# B&R Automation Studio project RobotComau
Automation Studio 4.11.2.75; technology packages: mapp 5.18.0, mappMotion 5.18.1, mappView 5.18.1, mappVision 5.18.0

## Configuration Config1

CPU 5APC3100.KBU1-000, AutomationRuntime B4.92, Build 4.1.2, Safety 0.0, Vc V4.72.5

### Task classes (Cpu.sw)
```
Cyclic#1 (cycle 2000 us, tolerance 0 us):
  Comau <- Comau.prg [disabled]
  OpcCtrl <- Sources.OpcCtrl.prg
  ComauManua <- PackML.PackML_Manual.prg
  PackML_Aut <- PackML.PackML_Auto.prg
  PackML_Log <- PackML.PackML_Logic.prg
  PackML_Sem <- PackML.PackML_SemiAuto.prg
  RobotMove <- (binary)
Cyclic#4:
  Alarms <- Alarms.prg
  Elements_d <- Elements_detection.prg
DataObjects: McAcpSys
NcDataObjects: McDriveLog
Binaries: McAcpDrv, udbdef, McAcpSim, mvLoader, arflatprv, McPathXT, TCData, visionUnit, mCoWebSc, McMechSys, FWRules, arcoal, arsvcreg, Settings, iomap, Config_3, Settings_1, viComp, Config_4, Role, ashwac, Hierarchy, asfw, Config_5, sysconf, Config_2, arconfig, Config_1, ashwd, User, Config_6, Config, Config_7, Config_9, PixelCount, Config_8, viApp, Matching15
Libraries: McBase, ViBase, AsZip, FileIO, AsARCfg, powerlnk, AsEPL, AsIO, sys_lib, astime, runtime, MpRobotics, McAxGroup, MpBase, McPathGen, McAxis, McProgInt, McAcpAx, CoTrace, standard, MpPackML, MpAlarmX, MpServer, MpUserX, asarprof, asieccon, asarlog, asmem, brsystem, dataobj, arssl, asopcuac, aseth, ashw, arcert, aruser
```

### Hardware
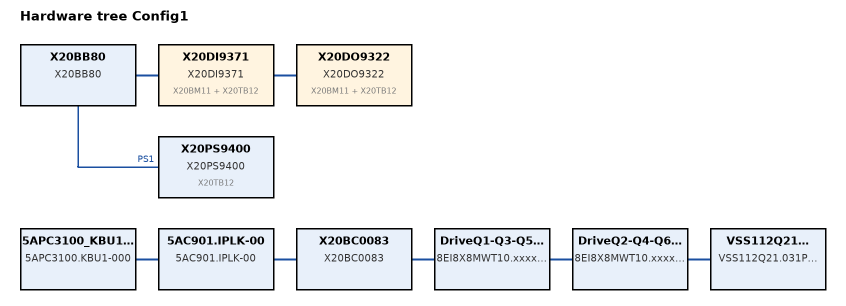
```
5AC901.IPLK-00 : 5AC901.IPLK-00 v1.8.0.1  [SL -> 5APC3100_KBU1_000.SL2]
  Connector IF1:
    MtuSize = 1500
    CycleTime = 400
    Channel1
    ChannelID1 = McAcpBroadcast
    ChannelType1 = OCTET[200]
    InternetAddress = 192.168.200.240
    SubnetMask = 255.255.255.0
5APC3100_KBU1_000 : 5APC3100.KBU1-000 v2.2.1.0
  Connector IF3:
    AssignedOperatingSystem = ARemb
    ActivateDevice = 1
    Mode = Manual
    InternetAddress = 192.168.0.10
    SubnetMask = 255.255.255.0
    ActivateSnmp = 2
  Connector IF4:
    AssignedOperatingSystem = ARemb
    ActivateDevice = 1
  Connector IF5:
    AssignedOperatingSystem = ARemb
  Connector IF6:
    AssignedOperatingSystem = ARemb
  Connector IF7:
    AssignedOperatingSystem = ARemb
  Connector IF8:
    AssignedOperatingSystem = ARemb
  ConfigurationID = RobotComau_Config1
  Simulation = 1
  RemMemDevice = PCI.2.IPLK.SRAM
  RemMemSize = 1024
  PermanentPvSize = 512
  RemanentGlobalPvSize = 512
  TimerDeviceType = EPLX2X
  TimerDevice = 5AC901.IPLK-00.IF1
  TaskClassIdleTime = 2000
  Cyclic1Duration = 2000
  Cyclic1Tolerance = 0
  FileDevice1
  FileDeviceName1 = CNC_PrgDir
  FileDevicePath1 = F:\RobotProgram
  FileDevice2
  FileDeviceName2 = F
  FileDevicePath2 = F:\
  FtpUser1
  FtpUsername1 = admin
  FtpUserPassword1 = QCzPEyxrRcQJkbJUmFYJydudCaTwVAMxyUFRcNQN44M=
  FtpUserSalt1 = 07CFXo9y
  FTPAccessRight1 = 0
  ActivateOpcUa = 1
  OpcUaInformationModels_PV_Version = 1
DriveQ1-Q3-Q5_Racer3_1 : 8EI8X8MWT10.xxxx-1 v2.3.1.1  [PLK1 -> X20BC0083.PLK2 (NodeNumber=4) [Cable Type=PowerlinkCable, Length=10, Version=1.0.0.3]; PLK2 -> DriveQ2-Q4-Q6_Racer3_1.PLK1 (NodeNumber=4) [Cable Type=PowerlinkCable, Length=10, Version=1.0.0.3]]
  DriveConfiguration/Module:
    McAcoposTypeID = AcoposP3TConfig
    ActivateACOPOSSimulationOnPLC = 0
  DriveConfiguration/Encoder/EncoderX41:
    InterfaceType = EnDat
  DriveConfiguration/Encoder/EncoderX42:
    InterfaceType = EnDat
  DriveConfiguration/Encoder/EncoderX43:
    InterfaceType = EnDat
  DriveConfiguration/Channel[1]/RealAxis:
    AxisReference = gAxisQ1_Racer3_1
    MechanicalElementsIsInvisible = 0
  DriveConfiguration/Channel[1]/RealAxis/MechanicalElements/Gearbox:
    InputIsReadOnly = 1
    Input = 81818
    OutputIsReadOnly = 1
    Output = 1000
  DriveConfiguration/Channel[1]/RealAxis/MechanicalElements/RotaryToLinearTransformation:
    ReferenceDistanceIsReadOnly = 1
    ReferenceDistance = 360
  DriveConfiguration/Channel[1]/RealAxis/Controller:
    ModeIsReadOnly = 1
    Mode = PositionControllerWithTorqueFeedForward
  DriveConfiguration/Channel[1]/RealAxis/Controller/Mode/Position:
    ProportionalGainIsReadOnly = 1
    ProportionalGain = 75.0
    IntegrationTimeIsReadOnly = 1
    IntegrationTime = 0.0
    TotalDelayTime = 0.0004
  DriveConfiguration/Channel[1]/RealAxis/Controller/Mode/Speed:
    ProportionalGainIsReadOnly = 1
    ProportionalGain = 2.0
    IntegrationTimeIsReadOnly = 1
    IntegrationTime = 0.0
    FilterTimeIsReadOnly = 1
    FilterTime = 0.0008
  DriveConfiguration/Channel[1]/RealAxis/Controller/Mode:
    FeedForwardIsReadOnly = 1
    FeedForward = CyclicValueFromAxesGroup
  DriveConfiguration/Channel[1]/RealAxis/Controller/Mode/LoopFilters:
    LoopFilterXIsReadOnly = 0
    LoopFilter1 = NotUsed
    LoopFilter2 = NotUsed
    LoopFilter3 = NotUsed
  DriveConfiguration/Channel[1]/RealAxis/Homing:
    ModeIsReadOnly = 0
    Mode = RestorePosition
    RestorePositionVariable = ::RestorePos[0]
  DriveConfiguration/Channel[1]/RealAxis/StopReaction:
    QuickstopIsReadOnly = 0
    Quickstop = DecelerationLimit
    DriveErrorIsReadOnly = 0
    DriveError = DecelerationLimit
  DriveConfiguration/Channel[1]/RealAxis/MovementErrorLimits:
    PositionError = 1.0
    VelocityErrorMonitoring = Automatic1
  DriveConfiguration/Channel[1]/RealAxis:
    JerkFilterIsReadOnly = 0
    JerkFilter = Used
  DriveConfiguration/Channel[1]/RealAxis/JerkFilter:
    JerkTimeMin = 0
    JerkTime = 0.01
  DriveConfiguration/Channel[1]/RealAxis/DigitalInputs/HomingSwitch:
    SourceIsReadOnly = 0
    Source = NotUsed
    Level = High
  DriveConfiguration/Channel[1]/RealAxis/DigitalInputs/PositiveLimitSwitch:
    SourceIsReadOnly = 0
    Source = NotUsed
    Level = High
  DriveConfiguration/Channel[1]/RealAxis/DigitalInputs/NegativeLimitSwitch:
    SourceIsReadOnly = 0
    Source = NotUsed
    Level = High
  DriveConfiguration/Channel[1]/RealAxis/DigitalInputs/Trigger1:
    Source = X8Trigger1
    Level = High
  DriveConfiguration/Channel[1]/RealAxis/DigitalInputs/Trigger2:
    Source = X8Trigger2
    Level = High
  DriveConfiguration/Channel[1]/RealAxis/DigitalInputs/Quickstop:
    Input = Trigger2
  DriveConfiguration/Channel[1]/RealAxis/Simulation:
    SimulationModeOnPLC = SetValueGeneration
    SimulationModeOnACOPOS = NotUsed
  DriveConfiguration/Channel[1]/RealAxis/AxisFeatures:
    FeatureRef[1] = Feature_Brake_Racer3_1
  DriveConfiguration/Channel[1]:
    ExternalEncoderAxis = NotUsed
  DriveConfiguration/Channel[2]/RealAxis:
    AxisReference = gAxisQ3_Racer3_1
    MechanicalElementsIsInvisible = 0
  DriveConfiguration/Channel[2]/RealAxis/MechanicalElements/Gearbox:
    InputIsReadOnly = 1
    Input = 72
    OutputIsReadOnly = 1
    Output = 1
  DriveConfiguration/Channel[2]/RealAxis/MechanicalElements/RotaryToLinearTransformation:
    ReferenceDistanceIsReadOnly = 1
    ReferenceDistance = 360
  DriveConfiguration/Channel[2]/RealAxis/Controller:
    ModeIsReadOnly = 1
    Mode = PositionControllerWithTorqueFeedForward
  DriveConfiguration/Channel[2]/RealAxis/Controller/Mode/Position:
    ProportionalGainIsReadOnly = 1
    ProportionalGain = 50.0
    IntegrationTimeIsReadOnly = 1
    IntegrationTime = 0.0
    TotalDelayTime = 0.0004
  DriveConfiguration/Channel[2]/RealAxis/Controller/Mode/Speed:
    ProportionalGainIsReadOnly = 1
    ProportionalGain = 1.5
    IntegrationTimeIsReadOnly = 1
    IntegrationTime = 0.0
    FilterTimeIsReadOnly = 1
    FilterTime = 0.0008
  DriveConfiguration/Channel[2]/RealAxis/Controller/Mode:
    FeedForwardIsReadOnly = 1
    FeedForward = CyclicValueFromAxesGroup
  DriveConfiguration/Channel[2]/RealAxis/Controller/Mode/LoopFilters:
    LoopFilterXIsReadOnly = 0
    LoopFilter1 = NotUsed
    LoopFilter2 = NotUsed
    LoopFilter3 = NotUsed
  DriveConfiguration/Channel[2]/RealAxis/Homing:
    ModeIsReadOnly = 0
    Mode = RestorePosition
    RestorePositionVariable = ::RestorePos[2]
  DriveConfiguration/Channel[2]/RealAxis/StopReaction:
    QuickstopIsReadOnly = 0
    Quickstop = DecelerationLimit
    DriveErrorIsReadOnly = 0
    DriveError = DecelerationLimit
  DriveConfiguration/Channel[2]/RealAxis/MovementErrorLimits:
    PositionError = 1.0
    VelocityErrorMonitoring = Automatic1
  DriveConfiguration/Channel[2]/RealAxis:
    JerkFilterIsReadOnly = 0
    JerkFilter = Used
  DriveConfiguration/Channel[2]/RealAxis/JerkFilter:
    JerkTimeMin = 0
    JerkTime = 0.01
  DriveConfiguration/Channel[2]/RealAxis/DigitalInputs/HomingSwitch:
    SourceIsReadOnly = 0
    Source = NotUsed
    Level = High
  DriveConfiguration/Channel[2]/RealAxis/DigitalInputs/PositiveLimitSwitch:
    SourceIsReadOnly = 0
    Source = NotUsed
    Level = High
  DriveConfiguration/Channel[2]/RealAxis/DigitalInputs/NegativeLimitSwitch:
    SourceIsReadOnly = 0
    Source = NotUsed
    Level = High
  DriveConfiguration/Channel[2]/RealAxis/DigitalInputs/Trigger1:
    Source = X8Trigger1
    Level = High
  DriveConfiguration/Channel[2]/RealAxis/DigitalInputs/Trigger2:
    Source = X8Trigger2
    Level = High
  DriveConfiguration/Channel[2]/RealAxis/DigitalInputs/Quickstop:
    Input = Trigger2
  DriveConfiguration/Channel[2]/RealAxis/Simulation:
    SimulationModeOnPLC = SetValueGeneration
    SimulationModeOnACOPOS = NotUsed
  DriveConfiguration/Channel[2]/RealAxis/AxisFeatures:
    FeatureRef[1] = Feature_Brake_Racer3_1
  DriveConfiguration/Channel[2]:
    ExternalEncoderAxis = NotUsed
  DriveConfiguration/Channel[3]/RealAxis:
    AxisReference = gAxisQ5_Racer3_1
    MechanicalElementsIsInvisible = 0
  DriveConfiguration/Channel[3]/RealAxis/MechanicalElements/Gearbox:
    InputIsReadOnly = 1
    Input = 612
    OutputIsReadOnly = 1
    Output = 10
  DriveConfiguration/Channel[3]/RealAxis/MechanicalElements/RotaryToLinearTransformation:
    ReferenceDistanceIsReadOnly = 1
    ReferenceDistance = 360
  DriveConfiguration/Channel[3]/RealAxis/Controller:
    ModeIsReadOnly = 1
    Mode = PositionControllerWithTorqueFeedForward
  DriveConfiguration/Channel[3]/RealAxis/Controller/Mode/Position:
    ProportionalGainIsReadOnly = 1
    ProportionalGain = 200.0
    IntegrationTimeIsReadOnly = 1
    IntegrationTime = 0.0
    TotalDelayTime = 0.0004
  DriveConfiguration/Channel[3]/RealAxis/Controller/Mode/Speed:
    ProportionalGainIsReadOnly = 1
    ProportionalGain = 1.5
    IntegrationTimeIsReadOnly = 1
    IntegrationTime = 0.0
    FilterTimeIsReadOnly = 1
    FilterTime = 0.0008
  DriveConfiguration/Channel[3]/RealAxis/Controller/Mode:
    FeedForwardIsReadOnly = 1
    FeedForward = CyclicValueFromAxesGroup
  DriveConfiguration/Channel[3]/RealAxis/Controller/Mode/LoopFilters:
    LoopFilterXIsReadOnly = 0
    LoopFilter1 = NotUsed
    LoopFilter2 = NotUsed
    LoopFilter3 = NotUsed
  DriveConfiguration/Channel[3]/RealAxis/Homing:
    ModeIsReadOnly = 0
    Mode = RestorePosition
    RestorePositionVariable = ::RestorePos[4]
  DriveConfiguration/Channel[3]/RealAxis/StopReaction:
    QuickstopIsReadOnly = 0
    Quickstop = DecelerationLimit
    DriveErrorIsReadOnly = 0
    DriveError = DecelerationLimit
  DriveConfiguration/Channel[3]/RealAxis/MovementErrorLimits:
    PositionError = 1.0
    VelocityErrorMonitoring = Automatic1
  DriveConfiguration/Channel[3]/RealAxis:
    JerkFilterIsReadOnly = 0
    JerkFilter = Used
  DriveConfiguration/Channel[3]/RealAxis/JerkFilter:
    JerkTimeMin = 0
    JerkTime = 0.01
  DriveConfiguration/Channel[3]/RealAxis/DigitalInputs/HomingSwitch:
    SourceIsReadOnly = 0
    Source = NotUsed
    Level = High
  DriveConfiguration/Channel[3]/RealAxis/DigitalInputs/PositiveLimitSwitch:
    SourceIsReadOnly = 0
    Source = NotUsed
    Level = High
  DriveConfiguration/Channel[3]/RealAxis/DigitalInputs/NegativeLimitSwitch:
    SourceIsReadOnly = 0
    Source = NotUsed
    Level = High
  DriveConfiguration/Channel[3]/RealAxis/DigitalInputs/Trigger1:
    Source = X8Trigger1
    Level = High
  DriveConfiguration/Channel[3]/RealAxis/DigitalInputs/Trigger2:
    Source = X8Trigger2
    Level = High
  DriveConfiguration/Channel[3]/RealAxis/DigitalInputs/Quickstop:
    Input = Trigger2
  DriveConfiguration/Channel[3]/RealAxis/Simulation:
    SimulationModeOnPLC = SetValueGeneration
    SimulationModeOnACOPOS = NotUsed
  DriveConfiguration/Channel[3]/RealAxis/AxisFeatures:
    FeatureRef[1] = Feature_Brake_Racer3_1
  DriveConfiguration/Channel[3]:
    ExternalEncoderAxis = NotUsed
DriveQ2-Q4-Q6_Racer3_1 : 8EI8X8MWT10.xxxx-1 v2.3.1.1  [PLK1 -> DriveQ1-Q3-Q5_Racer3_1.PLK2 (NodeNumber=5) [Cable Type=PowerlinkCable, Length=10, Version=1.0.0.3]; PLK2 -> VSS112Q21.031P-000.PLK2 (NodeNumber=5) [Cable Type=PowerlinkCable, Length=10, Version=1.0.0.3]]
  DriveConfiguration/Module:
    McAcoposTypeID = AcoposP3TConfig
    ActivateACOPOSSimulationOnPLC = 0
  DriveConfiguration/Encoder/EncoderX41:
    InterfaceType = EnDat
  DriveConfiguration/Encoder/EncoderX42:
    InterfaceType = EnDat
  DriveConfiguration/Encoder/EncoderX43:
    InterfaceType = EnDat
  DriveConfiguration/Channel[1]/RealAxis:
    AxisReference = gAxisQ2_Racer3_1
    MechanicalElementsIsInvisible = 0
  DriveConfiguration/Channel[1]/RealAxis/MechanicalElements/Gearbox:
    InputIsReadOnly = 1
    Input = 80
    OutputIsReadOnly = 1
    Output = 1
  DriveConfiguration/Channel[1]/RealAxis/MechanicalElements/RotaryToLinearTransformation:
    ReferenceDistanceIsReadOnly = 1
    ReferenceDistance = 360
  DriveConfiguration/Channel[1]/RealAxis/Controller:
    ModeIsReadOnly = 1
    Mode = PositionControllerWithTorqueFeedForward
  DriveConfiguration/Channel[1]/RealAxis/Controller/Mode/Position:
    ProportionalGainIsReadOnly = 1
    ProportionalGain = 50.0
    IntegrationTimeIsReadOnly = 1
    IntegrationTime = 0.0
    TotalDelayTime = 0.0004
  DriveConfiguration/Channel[1]/RealAxis/Controller/Mode/Speed:
    ProportionalGainIsReadOnly = 1
    ProportionalGain = 2.0
    IntegrationTimeIsReadOnly = 1
    IntegrationTime = 0.0
    FilterTimeIsReadOnly = 1
    FilterTime = 0.0008
  DriveConfiguration/Channel[1]/RealAxis/Controller/Mode:
    FeedForwardIsReadOnly = 1
    FeedForward = CyclicValueFromAxesGroup
  DriveConfiguration/Channel[1]/RealAxis/Controller/Mode/LoopFilters:
    LoopFilterXIsReadOnly = 0
    LoopFilter1 = NotUsed
    LoopFilter2 = NotUsed
    LoopFilter3 = NotUsed
  DriveConfiguration/Channel[1]/RealAxis/Homing:
    ModeIsReadOnly = 0
    Mode = RestorePosition
    RestorePositionVariable = ::RestorePos[1]
  DriveConfiguration/Channel[1]/RealAxis/StopReaction:
    QuickstopIsReadOnly = 0
    Quickstop = DecelerationLimit
    DriveErrorIsReadOnly = 0
    DriveError = DecelerationLimit
  DriveConfiguration/Channel[1]/RealAxis/MovementErrorLimits:
    PositionError = 1.0
    VelocityErrorMonitoring = Automatic1
  DriveConfiguration/Channel[1]/RealAxis:
    JerkFilterIsReadOnly = 0
    JerkFilter = Used
  DriveConfiguration/Channel[1]/RealAxis/JerkFilter:
    JerkTimeMin = 0
    JerkTime = 0.01
  DriveConfiguration/Channel[1]/RealAxis/DigitalInputs/HomingSwitch:
    SourceIsReadOnly = 0
    Source = NotUsed
    Level = High
  DriveConfiguration/Channel[1]/RealAxis/DigitalInputs/PositiveLimitSwitch:
    SourceIsReadOnly = 0
    Source = NotUsed
    Level = High
  DriveConfiguration/Channel[1]/RealAxis/DigitalInputs/NegativeLimitSwitch:
    SourceIsReadOnly = 0
    Source = NotUsed
    Level = High
  DriveConfiguration/Channel[1]/RealAxis/DigitalInputs/Trigger1:
    Source = X8Trigger1
    Level = High
  DriveConfiguration/Channel[1]/RealAxis/DigitalInputs/Trigger2:
    Source = X8Trigger2
    Level = High
  DriveConfiguration/Channel[1]/RealAxis/DigitalInputs/Quickstop:
    Input = Trigger2
  DriveConfiguration/Channel[1]/RealAxis/Simulation:
    SimulationModeOnPLC = SetValueGeneration
    SimulationModeOnACOPOS = NotUsed
  DriveConfiguration/Channel[1]/RealAxis/AxisFeatures:
    FeatureRef[1] = Feature_Brake_Racer3_1
  DriveConfiguration/Channel[1]:
    ExternalEncoderAxis = NotUsed
  DriveConfiguration/Channel[2]/RealAxis:
    AxisReference = gAxisQ4_Racer3_1
    MechanicalElementsIsInvisible = 0
  DriveConfiguration/Channel[2]/RealAxis/MechanicalElements/Gearbox:
    InputIsReadOnly = 1
    Input = 612
    OutputIsReadOnly = 1
    Output = 10
  DriveConfiguration/Channel[2]/RealAxis/MechanicalElements/RotaryToLinearTransformation:
    ReferenceDistanceIsReadOnly = 1
    ReferenceDistance = 360
  DriveConfiguration/Channel[2]/RealAxis/Controller:
    ModeIsReadOnly = 1
    Mode = PositionControllerWithTorqueFeedForward
  DriveConfiguration/Channel[2]/RealAxis/Controller/Mode/Position:
    ProportionalGainIsReadOnly = 1
    ProportionalGain = 100.0
    IntegrationTimeIsReadOnly = 1
    IntegrationTime = 0.0
    TotalDelayTime = 0.0004
  DriveConfiguration/Channel[2]/RealAxis/Controller/Mode/Speed:
    ProportionalGainIsReadOnly = 1
    ProportionalGain = 2.0
    IntegrationTimeIsReadOnly = 1
    IntegrationTime = 0.0
    FilterTimeIsReadOnly = 1
    FilterTime = 0.0008
  DriveConfiguration/Channel[2]/RealAxis/Controller/Mode:
    FeedForwardIsReadOnly = 1
    FeedForward = CyclicValueFromAxesGroup
  DriveConfiguration/Channel[2]/RealAxis/Controller/Mode/LoopFilters:
    LoopFilterXIsReadOnly = 0
    LoopFilter1 = NotUsed
    LoopFilter2 = NotUsed
    LoopFilter3 = NotUsed
  DriveConfiguration/Channel[2]/RealAxis/Homing:
    ModeIsReadOnly = 0
    Mode = RestorePosition
    RestorePositionVariable = ::RestorePos[3]
  DriveConfiguration/Channel[2]/RealAxis/StopReaction:
    QuickstopIsReadOnly = 0
    Quickstop = DecelerationLimit
    DriveErrorIsReadOnly = 0
    DriveError = DecelerationLimit
  DriveConfiguration/Channel[2]/RealAxis/MovementErrorLimits:
    PositionError = 1.0
    VelocityErrorMonitoring = Automatic1
  DriveConfiguration/Channel[2]/RealAxis:
    JerkFilterIsReadOnly = 0
    JerkFilter = Used
  DriveConfiguration/Channel[2]/RealAxis/JerkFilter:
    JerkTimeMin = 0
    JerkTime = 0.01
  DriveConfiguration/Channel[2]/RealAxis/DigitalInputs/HomingSwitch:
    SourceIsReadOnly = 0
    Source = NotUsed
    Level = High
  DriveConfiguration/Channel[2]/RealAxis/DigitalInputs/PositiveLimitSwitch:
    SourceIsReadOnly = 0
    Source = NotUsed
    Level = High
  DriveConfiguration/Channel[2]/RealAxis/DigitalInputs/NegativeLimitSwitch:
    SourceIsReadOnly = 0
    Source = NotUsed
    Level = High
  DriveConfiguration/Channel[2]/RealAxis/DigitalInputs/Trigger1:
    Source = X8Trigger1
    Level = High
  DriveConfiguration/Channel[2]/RealAxis/DigitalInputs/Trigger2:
    Source = X8Trigger2
    Level = High
  DriveConfiguration/Channel[2]/RealAxis/DigitalInputs/Quickstop:
    Input = Trigger2
  DriveConfiguration/Channel[2]/RealAxis/Simulation:
    SimulationModeOnPLC = SetValueGeneration
    SimulationModeOnACOPOS = NotUsed
  DriveConfiguration/Channel[2]/RealAxis/AxisFeatures:
    FeatureRef[1] = Feature_Brake_Racer3_1
  DriveConfiguration/Channel[2]:
    ExternalEncoderAxis = NotUsed
  DriveConfiguration/Channel[3]/RealAxis:
    AxisReference = gAxisQ6_Racer3_1
    MechanicalElementsIsInvisible = 0
  DriveConfiguration/Channel[3]/RealAxis/MechanicalElements/Gearbox:
    InputIsReadOnly = 1
    Input = 40
    OutputIsReadOnly = 1
    Output = 1
  DriveConfiguration/Channel[3]/RealAxis/MechanicalElements/RotaryToLinearTransformation:
    ReferenceDistanceIsReadOnly = 1
    ReferenceDistance = 360
  DriveConfiguration/Channel[3]/RealAxis/Controller:
    ModeIsReadOnly = 1
    Mode = PositionControllerWithTorqueFeedForward
  DriveConfiguration/Channel[3]/RealAxis/Controller/Mode/Position:
    ProportionalGainIsReadOnly = 1
    ProportionalGain = 200.0
    IntegrationTimeIsReadOnly = 1
    IntegrationTime = 0.0
    TotalDelayTime = 0.0004
  DriveConfiguration/Channel[3]/RealAxis/Controller/Mode/Speed:
    ProportionalGainIsReadOnly = 1
    ProportionalGain = 1.5
    IntegrationTimeIsReadOnly = 1
    IntegrationTime = 0.0
    FilterTimeIsReadOnly = 1
    FilterTime = 0.0008
  DriveConfiguration/Channel[3]/RealAxis/Controller/Mode:
    FeedForwardIsReadOnly = 1
    FeedForward = CyclicValueFromAxesGroup
  DriveConfiguration/Channel[3]/RealAxis/Controller/Mode/LoopFilters:
    LoopFilterXIsReadOnly = 0
    LoopFilter1 = NotUsed
    LoopFilter2 = NotUsed
    LoopFilter3 = NotUsed
  DriveConfiguration/Channel[3]/RealAxis/Homing:
    ModeIsReadOnly = 0
    Mode = RestorePosition
    RestorePositionVariable = ::RestorePos[5]
  DriveConfiguration/Channel[3]/RealAxis/StopReaction:
    QuickstopIsReadOnly = 0
    Quickstop = DecelerationLimit
    DriveErrorIsReadOnly = 0
    DriveError = DecelerationLimit
  DriveConfiguration/Channel[3]/RealAxis/MovementErrorLimits:
    PositionError = 1.0
    VelocityErrorMonitoring = Automatic1
  DriveConfiguration/Channel[3]/RealAxis:
    JerkFilterIsReadOnly = 0
    JerkFilter = Used
  DriveConfiguration/Channel[3]/RealAxis/JerkFilter:
    JerkTimeMin = 0
    JerkTime = 0.01
  DriveConfiguration/Channel[3]/RealAxis/DigitalInputs/HomingSwitch:
    SourceIsReadOnly = 0
    Source = NotUsed
    Level = High
  DriveConfiguration/Channel[3]/RealAxis/DigitalInputs/PositiveLimitSwitch:
    SourceIsReadOnly = 0
    Source = NotUsed
    Level = High
  DriveConfiguration/Channel[3]/RealAxis/DigitalInputs/NegativeLimitSwitch:
    SourceIsReadOnly = 0
    Source = NotUsed
    Level = High
  DriveConfiguration/Channel[3]/RealAxis/DigitalInputs/Trigger1:
    Source = X8Trigger1
    Level = High
  DriveConfiguration/Channel[3]/RealAxis/DigitalInputs/Trigger2:
    Source = X8Trigger2
    Level = High
  DriveConfiguration/Channel[3]/RealAxis/DigitalInputs/Quickstop:
    Input = Trigger2
  DriveConfiguration/Channel[3]/RealAxis/Simulation:
    SimulationModeOnPLC = SetValueGeneration
    SimulationModeOnACOPOS = NotUsed
  DriveConfiguration/Channel[3]/RealAxis/AxisFeatures:
    FeatureRef[1] = Feature_Brake_Racer3_1
  DriveConfiguration/Channel[3]:
    ExternalEncoderAxis = NotUsed
VSS112Q21.031P-000 : VSS112Q21.031P-000 v1.6.0.543  [PLK2 -> DriveQ2-Q4-Q6_Racer3_1.PLK2 (NodeNumber=6) [Cable Type=PowerlinkCable, Length=10, Version=1.0.0.3]]
  VisionConfig = gCamera
X20BB80 : X20BB80 v1.1.0.0
X20BC0083 : X20BC0083 v2.12.0.0  [PLK1 -> 5AC901.IPLK-00.IF1 (NodeNumber=3) [Cable Type=PowerlinkCable, Length=10, Version=1.0.0.3]; PLK2 -> DriveQ1-Q3-Q5_Racer3_1.PLK1 (NodeNumber=3) [Cable Type=PowerlinkCable, Length=10, Version=1.0.0.3]; SL -> X20BB80.SL1]
X20BM11 : X20BM11 v1.1.0.0  [X2X1 -> X20BB80.IF1]
X20BM11a : X20BM11 v1.1.0.0  [X2X1 -> X20BM11.X2X2]
X20DI9371 : X20DI9371 v1.3.0.0  [SS1 -> X20TB12a.SS; SL -> X20BM11.SL1]
X20DO9322 : X20DO9322 v1.4.0.0  [SS1 -> X20TB12b.SS; SL -> X20BM11a.SL1]
X20PS9400 : X20PS9400 v1.7.0.0  [SS1 -> X20TB12.SS; PS -> X20BB80.PS1]
X20TB12 : X20TB12 v1.0.0.0
X20TB12a : X20TB12 v1.0.0.0
X20TB12b : X20TB12 v1.0.0.0
```

### IoMap.iom - 5APC3100_KBU1_000/IoMap.iom
```iecst
VAR_CONFIG
	::Elements_d:Camera_0.ImageAcq AT %QX."VSS112Q21.031P-000".ImageAcquisition;
	::Elements_d:Camera_0.PixelCntSquareArray[0] AT %ID."VSS112Q21.031P-000".FoundedPixelsNum01;
	::Elements_d:Camera_0.PixelCntSquareArray[1] AT %ID."VSS112Q21.031P-000".FoundedPixelsNum02;
	::Elements_d:Camera_0.PixelCntSquareArray[2] AT %ID."VSS112Q21.031P-000".FoundedPixelsNum03;
	::Elements_d:Camera_0.PixelCntSquareArray[3] AT %ID."VSS112Q21.031P-000".FoundedPixelsNum04;
	::Elements_d:Camera_0.PixelCntSquareArray[4] AT %ID."VSS112Q21.031P-000".FoundedPixelsNum05;
	::Elements_d:Camera_0.PixelCntSquareArray[5] AT %ID."VSS112Q21.031P-000".FoundedPixelsNum06;
	::Elements_d:Camera_0.PixelCntSquareArray[6] AT %ID."VSS112Q21.031P-000".FoundedPixelsNum07;
	::Elements_d:Camera_0.PixelCntSquareArray[7] AT %ID."VSS112Q21.031P-000".FoundedPixelsNum08;
	::Elements_d:Camera_0.PixelCntSquareArray[8] AT %ID."VSS112Q21.031P-000".FoundedPixelsNum09;
	::Elements_d:Camera_0.PixelCntSquareArray[9] AT %ID."VSS112Q21.031P-000".FoundedPixelsNum10;
	::Elements_d:Camera_0.PixelCntSquareArray[10] AT %ID."VSS112Q21.031P-000".FoundedPixelsNum11;
	::Elements_d:Camera_0.PixelCntSquareArray[11] AT %ID."VSS112Q21.031P-000".FoundedPixelsNum12;
	::Elements_d:Camera_0.PixelCntSquareArray[12] AT %ID."VSS112Q21.031P-000".FoundedPixelsNum13;
	::Elements_d:Camera_0.PixelCntSquareArray[13] AT %ID."VSS112Q21.031P-000".FoundedPixelsNum14;
	::Elements_d:Camera_0.Focus AT %QW."VSS112Q21.031P-000".SetFocus;
	::Elements_d:Camera_0.ExposureTime AT %QD."VSS112Q21.031P-000".ExposureTime01;
	::Elements_d:Camera_0.Enable AT %QX."VSS112Q21.031P-000".EnableVF1;
	::Elements_d:Camera_0.NumSearch AT %QB."VSS112Q21.031P-000".NumSearch;
	::Elements_d:Camera_0.Ready AT %IX."VSS112Q21.031P-000".ImageAcquisitionReady;
	::Elements_d:Camera_0.FlashColor AT %QB."VSS112Q21.031P-000".FlashColor01;
	::Elements_d:Camera_0.FlashSegment AT %QB."VSS112Q21.031P-000".FlashSegment01;
	::Elements_d:Camera_0.ModelNumArray[0] AT %IB."VSS112Q21.031P-000".ModelNum01;
	::Elements_d:Camera_0.ModelNumArray[1] AT %IB."VSS112Q21.031P-000".ModelNum02;
	::Elements_d:Camera_0.ModelNumArray[2] AT %IB."VSS112Q21.031P-000".ModelNum03;
	::Elements_d:Camera_0.ModelNumArray[3] AT %IB."VSS112Q21.031P-000".ModelNum04;
	::Elements_d:Camera_0.ModelNumArray[4] AT %IB."VSS112Q21.031P-000".ModelNum05;
	::Elements_d:Camera_0.ModelNumArray[5] AT %IB."VSS112Q21.031P-000".ModelNum06;
	::Elements_d:Camera_0.ModelNumArray[6] AT %IB."VSS112Q21.031P-000".ModelNum07;
	::Elements_d:Camera_0.ModelNumArray[7] AT %IB."VSS112Q21.031P-000".ModelNum08;
	::Elements_d:Camera_0.ModelNumArray[8] AT %IB."VSS112Q21.031P-000".ModelNum09;
	::Elements_d:Camera_0.ModelNumArray[9] AT %IB."VSS112Q21.031P-000".ModelNum10;
	::Elements_d:Camera_0.ModelNumArray[10] AT %IB."VSS112Q21.031P-000".ModelNum11;
	::Elements_d:Camera_0.ModelNumArray[11] AT %IB."VSS112Q21.031P-000".ModelNum12;
	::Elements_d:Camera_0.ModelNumArray[12] AT %IB."VSS112Q21.031P-000".ModelNum13;
	::Elements_d:Camera_0.ModelNumArray[13] AT %IB."VSS112Q21.031P-000".ModelNum14;
	::doMagnet AT %QX."X20DO9322".DigitalOutput05;
END_VAR
```

### Config_1.axesgroup - 5APC3100_KBU1_000/mappMotion/Comau_Racer3_1/Config_1.axesgroup
```
Element gAxesGroup_Racer3_1 (Type=axesgroup)
  Type = PathGenAxesGroup
    ProcessingTaskClass = 255
    License = 1
    PhysicalAxes:
      JointAxes:
        JointAxisAxisRefIsReadOnly = 0
        JointAxis[1]:
          Name = Q1
          AxisRef = gAxisQ1_Racer3_1
        JointAxis[2]:
          Name = Q2
          AxisRef = gAxisQ2_Racer3_1
        JointAxis[3]:
          Name = Q3
          AxisRef = gAxisQ3_Racer3_1
        JointAxis[4]:
          Name = Q4
          AxisRef = gAxisQ4_Racer3_1
        JointAxis[5]:
          Name = Q5
          AxisRef = gAxisQ5_Racer3_1
        JointAxis[6]:
          Name = Q6
          AxisRef = gAxisQ6_Racer3_1
    MechanicalSystem:
      MechSysRefIsReadOnly = 0
      MechSysRef = MechSys_Racer3_1
    BasicSettings:
      ModalDataBehaviour = ResetToDefault
      GeometryPlanning:
        TCPResolutionIsReadOnly = 0
        TCPResolution:
          LengthResolution = 0.001
          AngleResolution = 0.001
        RoundingMode = Standard
        MaxCornerDeviation = 0.0
        MaxTangentialTransitionDeviation = 0.05
        MaxRadiusDeviation = 0.001
        WorkingPlane = XY
      TrajectoryPlanningIsReadOnly = 0
      TrajectoryPlanning = Basic
        LimitCheckResolutionIsReadOnly = 0
        LimitCheckResolution = UserDefinedTime
          TimeIsReadOnly = 0
          Time = 0.005
        BufferTime = UserDefinedTime
          Time = 0.050
      Miscellaneous:
        NonMovementsLimit = NotUsed
    AxesGroupFeatures:
      FeatureRef[1] = Feature_Programs_Racer3_1
      FeatureRef[2] = Feature_FeedForward_Racer3_1
      FeatureRef[3] = Feature_Jogging_Racer3_1
      FeatureRef[4] = Feature_SharedBrakesSignals_Racer3_1
      FeatureRef[5] = Feature_WorkspaceMonitoring
  Alarms = None
```

### Config_2.axis - 5APC3100_KBU1_000/mappMotion/Comau_Racer3_1/Config_2.axis
```
Element gAxisQ1_Racer3_1 (Type=axis)
  BaseTypeIsReadOnly = 1
  BaseType = RotaryBounded
    MeasurementUnitIsReadOnly = 1
    MeasurementUnit = 17476
    MeasurementResolutionIsReadOnly = 1
    MeasurementResolution = 0.001
    CountDirectionIsReadOnly = 1
    CountDirection = Inverse
  MovementLimitsIsReadOnly = 1
  MovementLimits = InternalForPathControlledAxis
    Position:
      LowerLimitMin = -170.0
      UpperLimitMax = 170.0
      LowerLimit = -170.0
      UpperLimit = 170.0
    VelocityIsReadOnly = 1
    Velocity:
      VelocityMax = 420.0
      Velocity = 420.0
    AccelerationIsReadOnly = 1
    Acceleration:
      AccelerationMax = 1100.0
      Acceleration = 1100.0
    DecelerationIsReadOnly = 1
    Deceleration:
      DecelerationMax = 1100.0
      Deceleration = 1100.0
    JerkIsReadOnly = 1
    Jerk = Basic
      JerkMax = 3.4E38
      Jerk = 11000.0
    TorqueIsInvisible = 0
  Alarms = None
Element gAxisQ2_Racer3_1 (Type=axis)
  BaseTypeIsReadOnly = 1
  BaseType = RotaryBounded
    MeasurementUnitIsReadOnly = 1
    MeasurementUnit = 17476
    MeasurementResolutionIsReadOnly = 1
    MeasurementResolution = 0.001
    CountDirectionIsReadOnly = 1
    CountDirection = Standard
  MovementLimitsIsReadOnly = 1
  MovementLimits = InternalForPathControlledAxis
    Position:
      LowerLimitMin = -95.0
      UpperLimitMax = 135.0
      LowerLimit = -95.0
      UpperLimit = 135.0
    VelocityIsReadOnly = 1
    Velocity:
      VelocityMax = 450.0
      Velocity = 450.0
    AccelerationIsReadOnly = 1
    Acceleration:
      AccelerationMax = 750.0
      Acceleration = 750.0
    DecelerationIsReadOnly = 1
    Deceleration:
      DecelerationMax = 750.0
      Deceleration = 750.0
    JerkIsReadOnly = 1
    Jerk = Basic
      JerkMax = 3.4E38
      Jerk = 7500.0
    TorqueIsInvisible = 0
  Alarms = None
Element gAxisQ3_Racer3_1 (Type=axis)
  BaseTypeIsReadOnly = 1
  BaseType = RotaryBounded
    MeasurementUnitIsReadOnly = 1
    MeasurementUnit = 17476
    MeasurementResolutionIsReadOnly = 1
    MeasurementResolution = 0.001
    CountDirectionIsReadOnly = 1
    CountDirection = Inverse
  MovementLimitsIsReadOnly = 1
  MovementLimits = InternalForPathControlledAxis
    Position:
      LowerLimitMin = -155.0
      UpperLimitMax = 90.0
      LowerLimit = -155.0
      UpperLimit = 90.0
    VelocityIsReadOnly = 1
    Velocity:
      VelocityMax = 480.0
      Velocity = 480.0
    AccelerationIsReadOnly = 1
    Acceleration:
      AccelerationMax = 1250.0
      Acceleration = 1250.0
    DecelerationIsReadOnly = 1
    Deceleration:
      DecelerationMax = 1250.0
      Deceleration = 1250.0
    JerkIsReadOnly = 1
    Jerk = Basic
      JerkMax = 3.4E38
      Jerk = 12500.0
    TorqueIsInvisible = 0
  Alarms = None
Element gAxisQ4_Racer3_1 (Type=axis)
  BaseTypeIsReadOnly = 1
  BaseType = RotaryBounded
    MeasurementUnitIsReadOnly = 1
    MeasurementUnit = 17476
    MeasurementResolutionIsReadOnly = 1
    MeasurementResolution = 0.001
    CountDirectionIsReadOnly = 1
    CountDirection = Standard
  MovementLimitsIsReadOnly = 1
  MovementLimits = InternalForPathControlledAxis
    Position:
      LowerLimitMin = -200.0
      UpperLimitMax = 200.0
      LowerLimit = -200.0
      UpperLimit = 200.0
    VelocityIsReadOnly = 1
    Velocity:
      VelocityMax = 600.0
      Velocity = 600.0
    AccelerationIsReadOnly = 1
    Acceleration:
      AccelerationMax = 1200.0
      Acceleration = 1200.0
    DecelerationIsReadOnly = 1
    Deceleration:
      DecelerationMax = 1200.0
      Deceleration = 1200.0
    JerkIsReadOnly = 1
    Jerk = Basic
      JerkMax = 3.4E38
      Jerk = 12000.0
    TorqueIsInvisible = 0
  Alarms = None
Element gAxisQ5_Racer3_1 (Type=axis)
  BaseTypeIsReadOnly = 1
  BaseType = RotaryBounded
    MeasurementUnitIsReadOnly = 1
    MeasurementUnit = 17476
    MeasurementResolutionIsReadOnly = 1
    MeasurementResolution = 0.001
    CountDirectionIsReadOnly = 1
    CountDirection = Standard
  MovementLimitsIsReadOnly = 1
  MovementLimits = InternalForPathControlledAxis
    Position:
      LowerLimitMin = -125.0
      UpperLimitMax = 125.0
      LowerLimit = -125.0
      UpperLimit = 125.0
    VelocityIsReadOnly = 1
    Velocity:
      VelocityMax = 600.0
      Velocity = 600.0
    AccelerationIsReadOnly = 1
    Acceleration:
      AccelerationMax = 1200.0
      Acceleration = 1200.0
    DecelerationIsReadOnly = 1
    Deceleration:
      DecelerationMax = 1200.0
      Deceleration = 1200.0
    JerkIsReadOnly = 1
    Jerk = Basic
      JerkMax = 3.4E38
      Jerk = 12000.0
    TorqueIsInvisible = 0
  Alarms = None
Element gAxisQ6_Racer3_1 (Type=axis)
  BaseTypeIsReadOnly = 1
  BaseType = RotaryBounded
    MeasurementUnitIsReadOnly = 1
    MeasurementUnit = 17476
    MeasurementResolutionIsReadOnly = 1
    MeasurementResolution = 0.001
    CountDirectionIsReadOnly = 1
    CountDirection = Standard
  MovementLimitsIsReadOnly = 1
  MovementLimits = InternalForPathControlledAxis
    Position:
      LowerLimitMin = -2700.0
      UpperLimitMax = 2700.0
      LowerLimit = -2700.0
      UpperLimit = 2700.0
    VelocityIsReadOnly = 1
    Velocity:
      VelocityMax = 875.0
      Velocity = 875.0
    AccelerationIsReadOnly = 1
    Acceleration:
      AccelerationMax = 1800.0
      Acceleration = 1800.0
    DecelerationIsReadOnly = 1
    Deceleration:
      DecelerationMax = 1800.0
      Deceleration = 1800.0
    JerkIsReadOnly = 1
    Jerk = Basic
      JerkMax = 3.4E38
      Jerk = 18000.0
    TorqueIsInvisible = 0
  Alarms = MpAlarmX
```

### Config_7.axesgroupfeature - 5APC3100_KBU1_000/mappMotion/Config_7.axesgroupfeature
```
Element Feature_WorkspaceMonitoring (Type=axesgroupfeature)
  Type = WorkspaceMonitoring
    ModalDataBehaviour = UseAxesGroupSettings
    WorkspaceRef = 
    SelfCollisionDetection = Enabled
    FlangeWorkspace = NotUsed
```

### Config.mpalarmxcore - 5APC3100_KBU1_000/mappServices/Config.mpalarmxcore
```
Element gAlarmXCore_0 (Type=mpalarmxcore)
  mapp.AlarmX.Core.Configuration:
    [0]:
      Name = HoldersHigh
      Message = Wykryto za dużo podstawek!
      Code = 101
      Behavior = LevelMonitoring
        Monitoring:
          MonitoredPV = ::Elements_d:DetectedHolders
          HighLimitEnable = Static
            Limit = 7
    [1]:
      Name = HoldersLow
      Message = Wykryto za mało podstawek!
      Code = 102
      Behavior = LevelMonitoring
        Monitoring:
          MonitoredPV = ::Elements_d:DetectedSquares
          LowLimitEnable = Static
            Limit = 7
```

### Config.mppackmlcore - 5APC3100_KBU1_000/mappServices/Config.mppackmlcore
```
Element gPackMLCore (Type=mppackmlcore)
  Core:
    StartupActiveMode = 1
    StartupActiveState = 2
  Modes:
    Mode[1]:
      ModeID = 1
      Name = Auto
      State[1] = 0
      State[5] = 0
      State[8] = 0
      State[9] = 0
      State[13] = 0
      State[14] = 0
    Mode[2]:
      ModeID = 2
      Name = Semiauto
    Mode[3]:
      ModeID = 3
```

### Config_14.mpaudittrail - 5APC3100_KBU1_000/mappServices/Config_14.mpaudittrail
```
Element gAuditTrail (Type=mpaudittrail)
  Audit:
    Events:
      [0] = 16
      [1] = 2
      [2] = 18
      [3] = 19
    TextSource = TXT
      Name = Audit/Event/Root
      Display = Ne
    Export:
      Encrypt = FALSE
  Alarms = MpAlarmX
```

### Config_2.mppackmlcore - 5APC3100_KBU1_000/mappServices/Config_2.mppackmlcore
```
Element gPackMLCore (Type=mppackmlcore)
  Modes:
    Mode[1]:
      ModeID = 1
      Name = Auto
    Mode[2]:
      ModeID = 2
      Name = Semiauto
    Mode[3]:
      ModeID = 3
```

### Config_8.mpalarmxcore - 5APC3100_KBU1_000/mappServices/Config_8.mpalarmxcore
```
Element gAlarmXCore0 (Type=mpalarmxcore)
  mapp.AlarmX.Core.Configuration:
    [0]:
      Name = SquaresAlarm
      Message = Za dużo podstawek
      Behavior = LevelMonitoring
        Monitoring:
          MonitoredPV = ::Elements_d:testAlarm
          LowLimitEnable = Static
            Limit = 6
          HighLimitEnable = Static
            Limit = 8
    [1]:
      Name = Error
      Message = ERROR
      Code = 1
      Behavior = LevelMonitoring
        Monitoring:
          MonitoredPV = ::Comau:MpRoboArm6Axis_0.Error
          HighLimitEnable = Static
            Limit = 1
```

## Configuration Config2

### Task classes (Cpu.sw)
```
Cyclic#1:
  Comau <- Comau.prg
  OpcCtrl <- Sources.OpcCtrl.prg
  ComauManua <- PackML.PackML_Manual.prg
  PackML_Aut <- PackML.PackML_Auto.prg
  PackML_Log <- PackML.PackML_Logic.prg
  RobotMove <- (binary)
Cyclic#4:
  Alarms <- Alarms.prg
  Elements_d <- Elements_detection.prg
  PackML_Sem <- PackML.PackML_SemiAuto.prg
DataObjects: McAcpSys
NcDataObjects: McDriveLog
Binaries: McAcpDrv, udbdef, McAcpSim, mvLoader, arflatprv, McPathXT, TCData, visionUnit, mCoWebSc, McMechSys, FWRules, arcoal, arsvcreg, viApp, Settings, iomap, Config_3, Settings_1, viComp, Config_4, Role, ashwac, Hierarchy, asfw, Config_5, sysconf, Config_2, arconfig, Config_1, ashwd, User, Config_6, Config, Config_7, Config_9, PixelCount, Config_8, Matching15
Libraries: McBase, ViBase, AsZip, FileIO, AsARCfg, powerlnk, AsEPL, AsIO, sys_lib, astime, runtime, MpRobotics, McAxGroup, MpBase, McPathGen, McAxis, McProgInt, McAcpAx, CoTrace, standard, MpPackML, MpAlarmX, MpServer, MpUserX, asarprof, asieccon, asarlog, asmem, brsystem, dataobj, arssl, asopcuac, aseth, ashw, arcert, aruser
```

## Logical view

Binary libraries used (declarations not repeated): operator, runtime, astime, AsIecCon, McBase, ViBase, AsZip, FileIO, AsARCfg, powerlnk, AsEPL, AsIO, sys_lib, MpRobotics, McAxGroup, MpBase, McPathGen, McAxis, McProgInt, McAcpAx, CoTrace, standard, MpPackML, AsOpcUac, MpAlarmX, MpServer, MpUserX, MpFile, AsBrStr

### Global.typ - Global data types
```iecst
TYPE
	gSafeType : 	STRUCT
		diEStop : BOOL;
		diEStopPanel : BOOL;
		diGuardDoor1 : BOOL;
		diGuardDoor2 : BOOL;
		EStop : BOOL;
		EStopPanel : BOOL;
		GuardingDoor : BOOL;
		SafeChannelOK1 : BOOL;
		SafeChannelOK2 : BOOL;
		doAcoposEnable1 : BOOL;
		doAcoposEnable2 : BOOL;
		CommunicationError : BOOL;
		ComErrorAck  : BOOL;

	END_STRUCT;
END_TYPE
```

### Global.var - Global variables
```iecst
VAR
	y : USINT;

	gSquareArray : ARRAY[0..13] OF BOOL; (*1 IF is square in i position*)
END_VAR
VAR RETAIN
	RestorePos : ARRAY[0..5] OF McAcpAxRestorePosType; (*Comau Home Position*)
END_VAR
VAR
	PZ : McPointType := (Pos:=(X:=435,Y:=0,Z:=685),Orient:=(Angle1:=0,Angle2:=90,Angle3:=0));
	pom : ARRAY[0..9] OF BOOL := [10(0)];
	P2up : McPointType := (Pos:=(X:=410,Y:=200,Z:=200),Orient:=(Angle1:=0,Angle2:=180,Angle3:=0));
	P2 : McPointType := (Pos:=(X:=410,Y:=200,Z:=140),Orient:=(Angle1:=0,Angle2:=180,Angle3:=0));
	P1up : McPointType := (Pos:=(X:=510,Y:=-300,Z:=200),Orient:=(Angle1:=0,Angle2:=180,Angle3:=0));
	P1 : McPointType := (Pos:=(X:=510,Y:=-300,Z:=140),Orient:=(Angle1:=0,Angle2:=180,Angle3:=0));
	P0 : McPointType := (Pos:=(X:=435,Y:=0,Z:=405),Orient:=(Angle1:=0,Angle2:=180,Angle3:=0));
	A : McAxisTargetType := (JointAxis:=[0,0,-90,0,90,0],SlaveAxis:=[100]);
	MpPackMLMode_SemiAuto : MpPackMLMode;
	MpPackMLMode_Manual : MpPackMLMode;
	MpPackMLMode_Auto : MpPackMLMode;
	MpPackMLCore_0 : MpPackMLCore;
	HOME : McPointType := (Pos:=(X:=435.9,Y:=0,Z:=685),Orient:=(Angle1:=0,Angle2:=90,Angle3:=0));
	gSafety : gSafeType;
	gRobPos : ARRAY[0..13] OF McPointType := [(Pos:=(X:=510,Y:=-300,Z:=70),Orient:=(Angle1:=0,Angle2:=180,Angle3:=0)),(Pos:=(X:=510,Y:=-200,Z:=140),Orient:=(Angle1:=0,Angle2:=180)),(Pos:=(X:=510,Y:=-100,Z:=140),Orient:=(Angle1:=0,Angle2:=180,Angle3:=0)),(Pos:=(X:=510,Y:=0,Z:=140),Orient:=(Angle1:=0,Angle2:=180,Angle3:=0)),(Pos:=(X:=510,Y:=100,Z:=140),Orient:=(Angle1:=0,Angle2:=180,Angle3:=0)),(Pos:=(X:=510,Y:=200,Z:=140),Orient:=(Angle1:=0,Angle2:=180)),(Pos:=(X:=510,Y:=300,Z:=140),Orient:=(Angle1:=0,Angle2:=180,Angle3:=0)),(Pos:=(X:=410,Y:=-300,Z:=140),Orient:=(Angle1:=0,Angle2:=180)),(Pos:=(X:=410,Y:=-200,Z:=140),Orient:=(Angle1:=0,Angle2:=180)),(Pos:=(X:=410,Y:=-100,Z:=140),Orient:=(Angle1:=0,Angle2:=180,Angle3:=0)),(Pos:=(X:=410,Y:=0,Z:=140),Orient:=(Angle1:=0,Angle2:=180,Angle3:=0)),(Pos:=(X:=410,Y:=100,Z:=140),Orient:=(Angle1:=0,Angle2:=180,Angle3:=0)),(Pos:=(X:=410,Y:=200,Z:=140),Orient:=(Angle1:=0,Angle2:=180,Angle3:=0)),(Pos:=(X:=410,Y:=300,Z:=140),Orient:=(Angle1:=0,Angle2:=180,Angle3:=0))];
	gIsPosGood : ARRAY[0..13] OF BOOL := [11(0),3(1)];
	gAimPos : ARRAY[0..13] OF INT := [11(0),1,2,3];
	gActPos : ARRAY[0..13] OF INT := [2(0),1,2(0),2,0,3,6(0)];
	gElementsArray : ARRAY[0..13] OF USINT;

END_VAR
```

### Package Logical/Libraries - Global libraries

- Visualisation Logical/mappView (not shown)

### Program Logical/Alarms (IEC)

#### Variables.var
```iecst
VAR
	MpAlarmXCore_0 : MpAlarmXCore;
END_VAR

VAR CONSTANT

END_VAR
```

#### Main.st
```iecst
PROGRAM _INIT
	MpAlarmXCore_0.MpLink := ADR(gAlarmXCore0);
	MpAlarmXCore_0.Enable := TRUE;

END_PROGRAM

PROGRAM _CYCLIC
	MpAlarmXCore_0();

END_PROGRAM

PROGRAM _EXIT
	MpAlarmXCore_0.Enable := FALSE;
	MpAlarmXCore_0();

END_PROGRAM
```

### Program Logical/Elements_detection (IEC)

#### Types.typ
```iecst
TYPE
	PixelCounterLimits : 	STRUCT
		WrenchLimit : UDINT;
		WasherBoltLimit : UDINT;
		ScrewLimit : UDINT;
	END_STRUCT;
	CameraStruct : 	STRUCT
		ExposureTime : UDINT := 30000;
		Focus : UINT := 30000;
		NumSearch : USINT;
		Enable : BOOL;
		diTrigger : BOOL;
		ImageAcq : BOOL;
		PixelCntSquareArray : ARRAY[0..13]OF UDINT;
		Ready : BOOL;
		FlashColor : USINT;
		ModelNumArray : ARRAY[0..13]OF USINT;
		FlashSegment : USINT;
	END_STRUCT;
END_TYPE
```

#### Variables.var
```iecst
VAR
	testAlarm : USINT;
	i : USINT;
	PixelRange_0 : PixelCounterLimits;
	DetectedSquares : USINT;
	Camera_0 : CameraStruct;
END_VAR
```

#### Main.st
```iecst
PROGRAM _INIT
	//CAMERA INITIAL VALUES
	Camera_0.Focus := 30000;
	Camera_0.ExposureTime := 40000;
	Camera_0.NumSearch := 14;
	Camera_0.Enable := 1;

	PixelRange_0.ScrewLimit := 200;
	PixelRange_0.WasherBoltLimit := 500;
	PixelRange_0.WrenchLimit := 2000;
	PixelRange_0.HolderLimit := 10000;

	///////////////////////////////
	DetectedSquares := 7;
	//////////////////////////////

END_PROGRAM

PROGRAM _CYCLIC
	//IMAGE ACQUISITION
	Camera_0.ImageAcq := Camera_0.diTrigger AND Camera_0.Ready;

	DetectedSquares := 0;

	FOR i := 0 TO 13 DO
		//SQUARES DETECTION
		gSquareArray[Camera_0.ModelNumArray[i]-1] := Camera_0.PixelCntSquareArray[i] < PixelRange_0.HolderLimit;
		IF Camera_0.PixelCntSquareArray[i] < PixelRange_0.HolderLimit THEN
			DetectedSquares := DetectedSquares + 1;
		END_IF

		IF Camera_0.PixelCntSquareArray[i] < 50 THEN
			//NOTHING
			gElementsArray[Camera_0.ModelNumArray[i]-1] := 0;
		ELSIF Camera_0.PixelCntSquareArray[i] < PixelRange_0.ScrewLimit THEN
			//SCREW
			//index nietestowy := 1
			gElementsArray[Camera_0.ModelNumArray[i]-1] := 1;
		ELSIF Camera_0.PixelCntSquareArray[i] < PixelRange_0.WasherBoltLimit THEN
			//WASHER BOLT
			//index nietestowy := 2
			gElementsArray[Camera_0.ModelNumArray[i]-1] := 2;
		ELSIF Camera_0.PixelCntSquareArray[i] < PixelRange_0.WrenchLimit THEN
			//WRENCH
			//index nietestowy := 4
			gElementsArray[Camera_0.ModelNumArray[i]-1] := 4;
		ELSE
			gElementsArray[Camera_0.ModelNumArray[i]-1] := 0;
		END_IF;

	END_FOR;

END_PROGRAM

PROGRAM _EXIT

END_PROGRAM
```

### Program Logical/PackML/PackML_Auto (IEC)

#### Main.st - Init, cyclic, exit code
```iecst
PROGRAM _INIT
	RestorePos;
	MpRoboArm6Axis_0.Enable := TRUE;

	MpRoboArm6Axis_0.Interrupt := 0;
	MpRoboArm6Axis_0.Continue := 0;

	MpRoboArm6Axis_0.Override  := 100.0;
	RoboParameters.CoordSystem := 0;
	RoboParameters.Velocity := 100;
	RoboParameters.Acceleration := 1000;
	RoboParameters.Deceleration := 1000;
	RoboParameters.ProgramName := 'Robotic.st';

END_PROGRAM

PROGRAM _CYCLIC
	Starting;
	Idle;
	Stopping;
	Resetting;
	Execute;
	Completing;
	Complete;
	Stopped;
	Holding;
	Held;
	Unhold;

	P2up;
	P2 ;
	P1up ;
	P1 ;
	P0;
	HOME;
	PZ;
	A;

	//throwing error
	IF MpRoboArm6Axis_0.Error THEN
		Step := ROBOTCTRL_ERROR;
		MpPackMLMode_Auto.Abort := TRUE;
	END_IF;

	IF diStop THEN
		MpRoboArm6Axis_0.Power := 0;
		MpPackMLMode_Auto.Stop := 1;
		diStop := 1;
		END_IF

	MpPackMLCore_0;
	MpPackMLMode_Auto;

	diStop;
	diStart;
	diReset;
	diExecute;
	cmdContinue;

	diAuto;
	diSemiAuto;
	diManual;

	MpRoboArm6Axis_0.MpLink     := ADR(gAxesGroup_Racer3_1);
	MpRoboArm6Axis_0.Parameters := ADR(RoboParameters);
	MpRoboArm6Axis_0.Override := 100.0;
	MpRoboArm6Axis_0.Enable := TRUE;
	MpRoboArm6Axis_0();

END_PROGRAM

PROGRAM _EXIT

END_PROGRAM
```

#### Variables.var - Local variables
```iecst
VAR
	diStop : BOOL; (*PackML Test*)
	diReset : BOOL; (*PackML Test*)
	diStart : BOOL; (*PackML Test*)
	diStopped : BOOL; (*PackML Test*)
	diIdle : BOOL; (*PackML Test*)
	diExecute : BOOL; (*PackML Test*)
	diCompleting : BOOL; (*PackML Test*)
	diComplete : BOOL; (*PackML Test*)
END_VAR
```

#### Stopped.st
```iecst
ACTION Stopped:
	IF MpPackMLStateIsActive(gPackMLCore,
		mpPACKML_STATE_STOPPED,
		1) THEN

		MpRoboArm6Axis_0.Power := FALSE;
		MpRoboArm6Axis_0.Stop := FALSE;
		diStop := 0;
		MpPackMLMode_Auto.Abort := 0;

		IF diReset THEN
			Step := ROBOTCTRL_POWER;
			MpPackMLMode_Auto.Reset := TRUE;
			diReset := FALSE;
		END_IF

	END_IF

END_ACTION
```

#### Resetting.st
```iecst
ACTION Resetting:

	IF MpPackMLStateIsActive(gPackMLCore,
		mpPACKML_STATE_RESETTING,
		1) THEN

		y := 0;

		CASE Step OF
			ROBOTCTRL_POWER:
				IF MpRoboArm6Axis_0.Info.ReadyToPowerOn THEN
					MpRoboArm6Axis_0.Power := TRUE;
					Step := ROBOTCTRL_WAIT_POWER;
				END_IF;

			ROBOTCTRL_WAIT_POWER:
				IF MpRoboArm6Axis_0.PowerOn THEN
					Step := ROBOTCTRL_HOME;
				END_IF;

			ROBOTCTRL_HOME:
				MpRoboArm6Axis_0.Home := TRUE;
				Step := ROBOTCTRL_WAIT_HOME;

			ROBOTCTRL_WAIT_HOME:
				IF MpRoboArm6Axis_0.IsHomed THEN
					MpRoboArm6Axis_0.Home := FALSE;
					Step := ROBOTCTRL_READY;
					MpPackMLStateComplete(gPackMLCore, 1);

				END_IF;

				END_CASE;

	END_IF;
END_ACTION
```

#### Idle.st
```iecst
ACTION Idle:

	IF MpPackMLStateIsActive(gPackMLCore,
		mpPACKML_STATE_IDLE,
		1) THEN

		MpPackMLMode_Auto.Reset := 0;

		CASE Step OF
			ROBOTCTRL_READY:
				MpRoboArm6Axis_0.MoveProgram := 0;

				IF NOT(MpRoboArm6Axis_0.PowerOn) THEN
					Step := ROBOTCTRL_DISABLED;
					MpPackMLMode_Auto.Stop := TRUE;
				END_IF;

				IF diStart THEN // diStart is active robot starts procedure
					diStart := FALSE;
					MpPackMLMode_Auto.Start := TRUE;
					Step := ROBOTCTRL_CHECK;
				END_IF;

		END_CASE;

	END_IF

END_ACTION
```

#### Starting.st
```iecst
ACTION Starting:

	IF MpPackMLStateIsActive(gPackMLCore,
		mpPACKML_STATE_STARTING,
		1) THEN

		MpPackMLMode_Auto.Start := 0;

		CASE Step OF
			ROBOTCTRL_CHECK: 	//checking if aim targets are available
				AimIsGood:=TRUE;
				FOR x:=0  TO SizeOfArray DO
					pom[0]:=1;
					IF gAimPos[x]>0 THEN
						pom[1]:=1;
						IF (gIsPosGood[x]=FALSE) THEN
							pom[2]:=1;
							Step:=ROBOTCTRL_ERROR_WRONG_AIM;
							AimIsGood:=0;
						END_IF;
					END_IF;
				END_FOR;
				IF AimIsGood=TRUE THEN
					y:=0;
					Step:=ROBOTCTRL_CALCULATE;
					MpPackMLStateComplete(gPackMLCore, 1);
				END_IF;

			ROBOTCTRL_ERROR_WRONG_AIM:
				//handling wrong target error
				IF diAck THEN
					diAck:=FALSE;
					Step:=ROBOTCTRL_CHECK;
				END_IF;

		END_CASE;

	END_IF
END_ACTION
```

#### Execute.st
```iecst
ACTION Execute:
	IF MpPackMLStateIsActive(gPackMLCore,
		mpPACKML_STATE_EXECUTE,
		1) THEN

		CASE Step OF
			ROBOTCTRL_CALCULATE:
				//checking if any move is needed and if all moves are done
				IF	P1P2_Ok THEN
					Step:=ROBOTCTRL_IS_MOVE_NEEDED;
				ELSIF y<IndexSize THEN
					Step:=ROBOTCTRL_CALCULATE_P1;
				ELSE
					diStart:=FALSE;
					Step:=ROBOTCTRL_READY;
					MpPackMLStateComplete(gPackMLCore, 1);
				END_IF;

			ROBOTCTRL_CALCULATE_P1:
				//assigning values to P1 and P1up
				FOR x:=0  TO SizeOfArray DO
					IF gActPos[x]=Index[y] THEN
						pom[3]:=1;
						P1.Orient.Angle1:=gRobPos[x].Orient.Angle1;
						P1.Orient.Angle2:=gRobPos[x].Orient.Angle2;
						P1.Orient.Angle3:=gRobPos[x].Orient.Angle3;
						P1.Pos.X:=gRobPos[x].Pos.X;
						P1.Pos.Y:=gRobPos[x].Pos.Y;
						P1.Pos.Z:=gRobPos[x].Pos.Z;
						P1up.Orient.Angle1:=gRobPos[x].Orient.Angle1;
						P1up.Orient.Angle2:=gRobPos[x].Orient.Angle2;
						P1up.Orient.Angle3:=gRobPos[x].Orient.Angle3;
						P1up.Pos.X:=gRobPos[x].Pos.X;
						P1up.Pos.Y:=gRobPos[x].Pos.Y;
						P1up.Pos.Z:=gRobPos[x].Pos.Z+50;

					END_IF;
				END_FOR;
				Step:=ROBOTCTRL_CALCULATE_P2;

			ROBOTCTRL_CALCULATE_P2:
				//assigning values to P2 and P2up
				FOR x:=0  TO SizeOfArray DO
					IF gAimPos[x]=Index[y] THEN
						pom[4]:=1;
						P2.Orient.Angle1:=gRobPos[x].Orient.Angle1;
						P2.Orient.Angle2:=gRobPos[x].Orient.Angle2;
						P2.Orient.Angle3:=gRobPos[x].Orient.Angle3;
						P2.Pos.X:=gRobPos[x].Pos.X;
						P2.Pos.Y:=gRobPos[x].Pos.Y;
						P2.Pos.Z:=gRobPos[x].Pos.Z;
						P2up.Orient.Angle1:=gRobPos[x].Orient.Angle1;
						P2up.Orient.Angle2:=gRobPos[x].Orient.Angle2;
						P2up.Orient.Angle3:=gRobPos[x].Orient.Angle3;
						P2up.Pos.X:=gRobPos[x].Pos.X;
						P2up.Pos.Y:=gRobPos[x].Pos.Y;
						P2up.Pos.Z:=gRobPos[x].Pos.Z+50;

					END_IF;
				END_FOR;
				P1P2_Ok:=1; // this flag means that new P1 and new P2 have been assigned
				Step:=ROBOTCTRL_CALCULATE;

			ROBOTCTRL_IS_MOVE_NEEDED:
				//checking if actual and aim positions are not the same
				IF P1.Orient.Angle1=P2.Orient.Angle1 AND P1.Pos.X=P2.Pos.X AND P1.Orient.Angle2=P2.Orient.Angle2 AND P1.Pos.Y=P2.Pos.Y AND P1.Orient.Angle3=P2.Orient.Angle3 AND P1.Pos.Z=P2.Pos.Z THEN
					y:=y+1; // index of next object
					P1P2_Ok:=0; // ready to assign new values to p1 p1up p2 p2up
					Step:=ROBOTCTRL_CALCULATE; // next assigning procedure with new object
				ELSE
					Step:=ROBOTCTRL_MOVE;   // going to move command
				END_IF;

			ROBOTCTRL_MOVE:
				IF cmdInterrupt OR MpRoboArm6Axis_0.MoveInterrupted THEN
					cmdInterrupt := FALSE;
					Step:=ROBOTCTRL_INTERRUPT;
					MpPackMLMode_Auto.Hold := 1;
				END_IF;

				//executing move procedure
				MpRoboArm6Axis_0.MoveProgram:=1;
				IF MpRoboArm6Axis_0.MoveDone THEN
					//retaking assigning procedure with new object after finishing move
					MpRoboArm6Axis_0.MoveProgram:=0;
					y:=y+1;
					P1P2_Ok:=0;
				 	Step:=ROBOTCTRL_CALCULATE;

				END_IF

		END_CASE;

	END_IF

END_ACTION
```

#### Completing.st
```iecst
ACTION Completing:
	IF MpPackMLStateIsActive(gPackMLCore,
		mpPACKML_STATE_COMPLETING,
		1) THEN

			MpPackMLStateComplete(gPackMLCore, 1);

	END_IF

END_ACTION
```

#### Complete.st
```iecst
ACTION Complete:
	IF MpPackMLStateIsActive(gPackMLCore,
		mpPACKML_STATE_COMPLETE,
		1) THEN

	//MpPackMLMode_Auto.Stop := 1;
		IF diReset THEN
			MpPackMLStateComplete(gPackMLCore, 1);
			MpPackMLMode_Auto.Reset := 1;
			diReset := 0;
			Step := ROBOTCTRL_POWER;

			END_IF;
	END_IF

END_ACTION
```

#### Stopping.st
```iecst
ACTION Stopping:
	IF MpPackMLStateIsActive(gPackMLCore,
		mpPACKML_STATE_STOPPING,
		1) THEN

		//STOP EVERYTHING
		MpRoboArm6Axis_0.Stop := TRUE;

		MpRoboArm6Axis_0.Power := FALSE;

		diStop := 0;

		IF NOT MpRoboArm6Axis_0.InMotion THEN
			MpPackMLStateComplete(gPackMLCore, 1);
			END_IF;

	END_IF

END_ACTION
```

#### Holding.st
```iecst
ACTION Holding:

	IF MpPackMLStateIsActive(gPackMLCore,
		mpPACKML_STATE_HOLDING,
		1) THEN

		MpRoboArm6Axis_0.Interrupt:=TRUE;
		IF MpRoboArm6Axis_0.MoveInterrupted THEN
			Step:=ROBOTCTRL_INTERRUPTING;
			MpPackMLStateComplete(gPackMLCore, 1);
		END_IF
	END_IF

END_ACTION
```

#### Held.st
```iecst
ACTION Held:

	IF MpPackMLStateIsActive(gPackMLCore,
		mpPACKML_STATE_HELD,
		1) THEN

		IF cmdContinue THEN
			cmdContinue:=FALSE;
			MpRoboArm6Axis_0.Interrupt:=FALSE;
			Step:=ROBOTCTRL_CONTINUE;
			MpPackMLMode_Auto.Unhold := 1;
		END_IF
	END_IF

END_ACTION
```

#### Unhold.st
```iecst
ACTION Unhold:

	IF MpPackMLStateIsActive(gPackMLCore,
		mpPACKML_STATE_UNHOLDING,
		1) THEN

		MpRoboArm6Axis_0.Continue := 1;
		MpPackMLMode_Auto.Unhold := 0;
		IF  MpRoboArm6Axis_0.InMotion THEN
			MpRoboArm6Axis_0.Continue:=0;
			Step:=ROBOTCTRL_MOVE;
			MpPackMLStateComplete(gPackMLCore, 1);
			MpPackMLMode_Auto.Hold := 0;
		END_IF
	END_IF

END_ACTION
```

#### Aborting.st - not listed in the package file held
```iecst
ACTION Aborting:

	IF MpPackMLStateIsActive(gPackMLCore,
		mpPACKML_STATE_ABORTING,
		1) THEN

		MpPackMLMode_Auto.Abort := 0;

		PackML_State := 'ABORTING';
		MpRoboArm6Axis_0.Power := FALSE;

		IF NOT MpRoboArm6Axis_0.PowerOn THEN
			MpPackMLStateComplete(gPackMLCore, 1);

			Step := ROBOTCTRL_POWER_OFF;
			Step_State := 'POWER_OFF';

		END_IF;
	END_IF

END_ACTION
```

### Program Logical/PackML/PackML_SemiAuto (IEC)

#### Main.st
```iecst
PROGRAM _INIT
	Step := ROBOTCTRL_POWER_OFF;

END_PROGRAM

PROGRAM _CYCLIC
	Starting;
	Idle;
	Stopping;
	Resetting;
	Execute;
	Completing;
	Complete;
	Stopped;

END_PROGRAM

PROGRAM _EXIT
	(* Insert code here *)

END_PROGRAM
```

### Program Logical/PackML/PackML_Manual (IEC)

#### Main.st
```iecst
PROGRAM _INIT
	(* Insert code here *)

END_PROGRAM

PROGRAM _CYCLIC
	Starting;
	Idle;
	Stopping;
	Resetting;
	Execute;
	Completing;
	Complete;
	Stopped;

	VelocityQ;
	doMagnet;

	RoboParameters.Jog.Velocity[0] := VelocityQ1;
	RoboParameters.Jog.Velocity[1] := VelocityQ2;
	RoboParameters.Jog.Velocity[2] := VelocityQ3;
	RoboParameters.Jog.Velocity[3] := VelocityQ4;
	RoboParameters.Jog.Velocity[4] := VelocityQ5;
	RoboParameters.Jog.Velocity[5] := VelocityQ6;

	IF cartezianVSjog THEN
		RoboParameters.Jog.CoordSystem := 10;
	ELSE
		RoboParameters.Jog.CoordSystem := 0;
	END_IF

	IF diManual THEN
		RoboParameters.ProgramName := 'HOME.st';
	ELSE
		RoboParameters.ProgramName := 'Robotic.st';
	END_IF

END_PROGRAM

PROGRAM _EXIT
	(* Insert code here *)

END_PROGRAM
```

### Variables.var - not listed in the package file held
```iecst
VAR
	Step : {REDUND_UNREPLICABLE} Step_typ := (0);

	diAuto : BOOL;
	diManual : BOOL;
	diSemiAuto : BOOL;
	MpRoboArm6Axis_0 : MpRoboArm6Axis;
	RoboParameters : MpRoboArm6AxisParType;

	x : INT := 0;
	AimIsGood : BOOL := FALSE;
	P1P2_Ok : BOOL := FALSE;

	diAck : BOOL;
	cmdInterrupt : BOOL;
	cmdContinue : BOOL;
	diStop : BOOL;
	diReset : BOOL;
	diStart : BOOL;
	diExecute : BOOL;

END_VAR

VAR CONSTANT
	SizeOfArray : INT := 13;
	IndexSize : INT := 3;
	Index : ARRAY[0..2] OF INT := [1,2,3];
END_VAR
```

### Main.st - not listed in the package file held
```iecst
PROGRAM _INIT
	(* Insert code here *)
	MpPackMLCore_0.MpLink := ADR(gPackMLCore);
	MpPackMLCore_0.Enable := TRUE;

	MpPackMLMode_0.MpLink := ADR(gPackMLCore);
	MpPackMLMode_0.Enable := TRUE;
	MpPackMLMode_0.ModeID := 1;
END_PROGRAM

PROGRAM _CYCLIC
	(* Insert code here *)
	MpPackMLCore_0();
	MpPackMLMode_0();
END_PROGRAM

PROGRAM _EXIT
	(* Insert code here *)

END_PROGRAM
```

### Program Logical/Comau (IEC)

#### Types.typ
```iecst
TYPE
	Step_typ :
		(
		ROBOTCTRL_DISABLED,
		ROBOTCTRL_POWER,
		ROBOTCTRL_WAIT_POWER,
		ROBOTCTRL_HOME,
		ROBOTCTRL_WAIT_HOME,
		ROBOTCTRL_READY,
		ROBOTCTRL_CALCULATE,
		ROBOTCTRL_CHECK,
		ROBOTCTRL_CALCULATE_P1,
		ROBOTCTRL_CALCULATE_P2,
		ROBOTCTRL_IS_MOVE_NEEDED,
		ROBOTCTRL_MOVE,
		ROBOTCTRL_ERROR_WRONG_AIM,
		ROBOTCTRL_ERROR,
		ROBOTCTRL_STOP,
		ROBOTCTRL_INTERRUPT,
			ROBOTCTRL_INTERRUPTING,
		ROBOTCTRL_CONTINUE,
		ROBOTCTRL_POWER_OFF,
		ROBOTCTRL_COMPLITE
		);
END_TYPE
```

#### Variables.var
```iecst
VAR
	TCPvalue : INT;
	manual : BOOL; (*Zalacza wybór trybu 0 - auto 1 - manual *)
	cartezianVSjog : BOOL; (*Wybór miedzy sterowaniem we wspólrzednych wewnetrznych - 0 / zewnętrznych - 1 *)
	MpRoboArm6Axis_0 : MpRoboArm6Axis;
	X1 : LREAL; (*wspólrzedna przekazywana do próbnego programu gdybysmy chcieli dojechac w okreslone miejsce*)
	Y1 : LREAL; (*wspólrzedna przekazywana do próbnego programu gdybysmy chcieli dojechac w okreslone miejsce*)
	Z1 : LREAL; (*wspólrzedna przekazywana do próbnego programu gdybysmy chcieli dojechac w okreslone miejsce*)
	A1 : LREAL; (*wspólrzedna przekazywana do próbnego programu gdybysmy chcieli dojechac w okreslone miejsce*)
	B1 : LREAL; (*wspólrzedna przekazywana do próbnego programu gdybysmy chcieli dojechac w okreslone miejsce*)
	C1 : LREAL; (*wspólrzedna przekazywana do próbnego programu gdybysmy chcieli dojechac w okreslone miejsce*)
	VelocityQ1 : REAL; (*Przypisanie predkosci do parametru 1 w zależnosci od wyboru wspólrzednych*)
	VelocityQ2 : REAL; (*Przypisanie predkosci do parametru 2 w zależnosci od wyboru wspólrzednych*)
	VelocityQ3 : REAL; (*Przypisanie predkosci do parametru 3 w zależnosci od wyboru wspólrzednych*)
	VelocityQ4 : REAL; (*Przypisanie predkosci do parametru 4 w zależnosci od wyboru wspólrzednych*)
	VelocityQ5 : REAL; (*Przypisanie predkosci do parametru 5 w zależnosci od wyboru wspólrzednych*)
	VelocityQ6 : REAL; (*Przypisanie predkosci do parametru 6 w zależnosci od wyboru wspólrzednych*)
	VelocityQ : REAL;
	doMagnet : BOOL;
	RoboParameters : MpRoboArm6AxisParType;
	x : INT := 0;
	AimIsGood : BOOL := FALSE;
	Step : {REDUND_UNREPLICABLE} Step_typ := (0);
	cmdTurnOn : BOOL := FALSE;
	cmdTurnOff : BOOL := FALSE;
	cmdExecute : BOOL := FALSE;
	P1P2_Ok : BOOL := FALSE;
	cmdAck : BOOL;
	cmdStop : BOOL;
	cmdStart : BOOL;
	cmdInterrupt : BOOL;
	cmdContinue : BOOL;
END_VAR
VAR CONSTANT
	SizeOfArray : INT := 13;
	IndexSize : INT := 3;
	Index : ARRAY[0..2] OF INT := [1,2,3];
END_VAR
```

#### Main.st
```iecst
PROGRAM _INIT
	RestorePos;
	MpRoboArm6Axis_0.Enable := TRUE;

	MpRoboArm6Axis_0.Override  := 100.0;
	RoboParameters.CoordSystem := 0;
	RoboParameters.Velocity := 100;
	RoboParameters.Acceleration := 1000;
	RoboParameters.Deceleration := 1000;
	RoboParameters.ProgramName := 'Robotic.st';
	x;

END_PROGRAM

PROGRAM _CYCLIC

	P2up;
	P2 ;
	P1up ;
	P1 ;
	P0;
	HOME;
	PZ;
	A;

	RoboParameters.Jog.Velocity[0] := VelocityQ1;
	RoboParameters.Jog.Velocity[1] := VelocityQ2;
	RoboParameters.Jog.Velocity[2] := VelocityQ3;
	RoboParameters.Jog.Velocity[3] := VelocityQ4;
	RoboParameters.Jog.Velocity[4] := VelocityQ5;
	RoboParameters.Jog.Velocity[5] := VelocityQ6;

	IF cartezianVSjog THEN
		RoboParameters.Jog.CoordSystem := 10;
	ELSE
		RoboParameters.Jog.CoordSystem := 0;
	END_IF

	IF manual THEN
		RoboParameters.ProgramName := 'HOME.st';
	ELSE
		RoboParameters.ProgramName := 'Robotic.st';
	END_IF
//throwing error
	IF MpRoboArm6Axis_0.Error THEN
		Step := ROBOTCTRL_ERROR;
	END_IF;
//turning off
	IF cmdTurnOff THEN
		cmdTurnOff := FALSE;
		Step:=ROBOTCTRL_POWER_OFF;
	END_IF;

	CASE Step OF

		ROBOTCTRL_DISABLED:
			IF cmdTurnOn THEN
				cmdTurnOn := FALSE;
				Step := ROBOTCTRL_POWER;
			END_IF;

		ROBOTCTRL_POWER:
			IF MpRoboArm6Axis_0.Info.ReadyToPowerOn THEN
				MpRoboArm6Axis_0.Power := TRUE;
				Step := ROBOTCTRL_WAIT_POWER;
			END_IF;

		ROBOTCTRL_WAIT_POWER:
			IF MpRoboArm6Axis_0.PowerOn THEN
				Step := ROBOTCTRL_HOME;
			END_IF;

		ROBOTCTRL_HOME:
			MpRoboArm6Axis_0.Home := TRUE;
			Step := ROBOTCTRL_WAIT_HOME;

		ROBOTCTRL_WAIT_HOME:
			IF MpRoboArm6Axis_0.IsHomed THEN
				MpRoboArm6Axis_0.Home := FALSE;
				Step := ROBOTCTRL_READY;
			END_IF;

		ROBOTCTRL_READY:
			MpRoboArm6Axis_0.MoveProgram:=0;
			IF cmdTurnOff THEN
				cmdTurnOff := FALSE;
			Step :=ROBOTCTRL_POWER_OFF;
			END_IF;

			IF NOT(MpRoboArm6Axis_0.PowerOn) THEN
				Step := ROBOTCTRL_DISABLED;
			END_IF;

			IF cmdExecute THEN
				cmdExecute:=FALSE;
				Step := ROBOTCTRL_CHECK; // if cmdexecute is active robot starts procedure

			END_IF;

		ROBOTCTRL_ERROR:
			// Error handling
			IF NOT(MpRoboArm6Axis_0.Error) THEN
				IF MpRoboArm6Axis_0.PowerOn THEN
					Step := ROBOTCTRL_READY;
				ELSE
					Step := ROBOTCTRL_DISABLED;
				END_IF;
			END_IF;

		ROBOTCTRL_CHECK: 	//checking if aim targets are available
			AimIsGood:=TRUE;
			FOR x:=0  TO SizeOfArray DO
				pom[0]:=1;
				IF gAimPos[x]>0 THEN
					pom[1]:=1;
					IF (gIsPosGood[x]=FALSE) THEN
						pom[2]:=1;
						Step:=ROBOTCTRL_ERROR_WRONG_AIM;
						AimIsGood:=0;
					END_IF;
				END_IF;
			END_FOR;
			IF AimIsGood=TRUE THEN
				y:=0;
				Step:=ROBOTCTRL_CALCULATE;
			END_IF;

		ROBOTCTRL_POWER_OFF:
			MpRoboArm6Axis_0.Power := FALSE;
			IF NOT MpRoboArm6Axis_0.PowerOn THEN
				Step:=ROBOTCTRL_DISABLED;
			END_IF

		ROBOTCTRL_CALCULATE:
			//checking if any move is needed and if all moves are done
			IF	P1P2_Ok THEN
				Step:=ROBOTCTRL_IS_MOVE_NEEDED;
			ELSIF y<IndexSize THEN
				Step:=ROBOTCTRL_CALCULATE_P1;
			ELSE
				cmdExecute:=FALSE;
				Step:=ROBOTCTRL_READY;
			END_IF;

		ROBOTCTRL_CALCULATE_P1:
			//assigning values to P1 and P1up
			FOR x:=0  TO SizeOfArray DO
				IF gActPos[x]=Index[y] THEN
					pom[3]:=1;
					P1.Orient.Angle1:=gRobPos[x].Orient.Angle1;
					P1.Orient.Angle2:=gRobPos[x].Orient.Angle2;
					P1.Orient.Angle3:=gRobPos[x].Orient.Angle3;
					P1.Pos.X:=gRobPos[x].Pos.X;
					P1.Pos.Y:=gRobPos[x].Pos.Y;
					P1.Pos.Z:=gRobPos[x].Pos.Z;
					P1up.Orient.Angle1:=gRobPos[x].Orient.Angle1;
					P1up.Orient.Angle2:=gRobPos[x].Orient.Angle2;
					P1up.Orient.Angle3:=gRobPos[x].Orient.Angle3;
					P1up.Pos.X:=gRobPos[x].Pos.X;
					P1up.Pos.Y:=gRobPos[x].Pos.Y;
					P1up.Pos.Z:=gRobPos[x].Pos.Z+100;

				END_IF;
			END_FOR;
			Step:=ROBOTCTRL_CALCULATE_P2;

		ROBOTCTRL_CALCULATE_P2:
			//assigning values to P2 and P2up
			FOR x:=0  TO SizeOfArray DO
				IF gAimPos[x]=Index[y] THEN
					pom[4]:=1;
					P2.Orient.Angle1:=gRobPos[x].Orient.Angle1;
					P2.Orient.Angle2:=gRobPos[x].Orient.Angle2;
					P2.Orient.Angle3:=gRobPos[x].Orient.Angle3;
					P2.Pos.X:=gRobPos[x].Pos.X;
					P2.Pos.Y:=gRobPos[x].Pos.Y;
					P2.Pos.Z:=gRobPos[x].Pos.Z;
					P2up.Orient.Angle1:=gRobPos[x].Orient.Angle1;
					P2up.Orient.Angle2:=gRobPos[x].Orient.Angle2;
					P2up.Orient.Angle3:=gRobPos[x].Orient.Angle3;
					P2up.Pos.X:=gRobPos[x].Pos.X;
					P2up.Pos.Y:=gRobPos[x].Pos.Y;
					P2up.Pos.Z:=gRobPos[x].Pos.Z+100;

				END_IF;
			END_FOR;
			P1P2_Ok:=1; // this flag means that new P1 and new P2 have been assigned
			Step:=ROBOTCTRL_CALCULATE;

		ROBOTCTRL_IS_MOVE_NEEDED:
			//checking if actual and aim positions are not the same
			IF P1.Orient.Angle1=P2.Orient.Angle1 AND P1.Pos.X=P2.Pos.X AND P1.Orient.Angle2=P2.Orient.Angle2 AND P1.Pos.Y=P2.Pos.Y AND P1.Orient.Angle3=P2.Orient.Angle3 AND P1.Pos.Z=P2.Pos.Z THEN
				y:=y+1;
				P1P2_Ok:=0;
				Step:=ROBOTCTRL_CALCULATE;
			ELSE
				Step:=ROBOTCTRL_MOVE;
			END_IF;

		ROBOTCTRL_MOVE:
			IF cmdInterrupt OR MpRoboArm6Axis_0.MoveInterrupted THEN
				cmdInterrupt := FALSE;
				Step:=ROBOTCTRL_INTERRUPT;
			END_IF;

			IF cmdStop OR MpRoboArm6Axis_0.Stopped THEN
				cmdStop := FALSE;
				Step:=ROBOTCTRL_STOP;

			END_IF;
			//executing move procedure
			MpRoboArm6Axis_0.MoveProgram:=1;
			IF MpRoboArm6Axis_0.MoveDone THEN
				MpRoboArm6Axis_0.MoveProgram:=0;
				y:=y+1;
				P1P2_Ok:=0;
				IF y=IndexSize THEN
					Step:=ROBOTCTRL_COMPLITE;
				ELSE
					Step:=ROBOTCTRL_CALCULATE;
				END_IF
			END_IF

		ROBOTCTRL_COMPLITE:
		Step:=ROBOTCTRL_POWER_OFF;

		ROBOTCTRL_INTERRUPT:
			MpRoboArm6Axis_0.Interrupt:=TRUE;
			IF MpRoboArm6Axis_0.MoveInterrupted THEN
				Step:=ROBOTCTRL_INTERRUPTING;
				END_IF

		ROBOTCTRL_INTERRUPTING:
			IF cmdContinue THEN
				cmdContinue:=FALSE;
				MpRoboArm6Axis_0.Interrupt:=FALSE;
				Step:=ROBOTCTRL_CONTINUE;
			END_IF

		ROBOTCTRL_CONTINUE:
			MpRoboArm6Axis_0.Continue:=1;
			IF  MpRoboArm6Axis_0.InMotion THEN
				MpRoboArm6Axis_0.Continue:=0;
				Step:=ROBOTCTRL_MOVE;
			END_IF

		ROBOTCTRL_STOP:
			MpRoboArm6Axis_0.Stop:=TRUE;
			IF MpRoboArm6Axis_0.Stopped THEN
				MpRoboArm6Axis_0.Stop:=FALSE;
				Step:=ROBOTCTRL_DISABLED;
				END_IF

		ROBOTCTRL_ERROR_WRONG_AIM:
			//handling wrong target error
			IF cmdAck THEN
				cmdAck:=FALSE;
				Step:=ROBOTCTRL_READY;
			END_IF;

	END_CASE;

	MpRoboArm6Axis_0.MpLink     := ADR(gAxesGroup_Racer3_1);
	MpRoboArm6Axis_0.Parameters := ADR(RoboParameters);
	MpRoboArm6Axis_0.Override := 100.0;
	MpRoboArm6Axis_0.Enable := TRUE;
	MpRoboArm6Axis_0();

END_PROGRAM

PROGRAM _EXIT

END_PROGRAM
```

### HOME.st
```iecst
VAR

	A : McAxisTargetType := (JointAxis:=[0, 0, -90, 0, 0, 0], SlaveAxis:=[100]);

END_VAR

	PROGRAM _MAIN

	Feedrate(2000);    //move with reduced speed
	MoveA(A); //move HOME
	END_PROGRAM
```

### Robotic.st
```iecst
VAR {AT PLC}
P2up : McPointType;
P2 : McPointType;
P1up : McPointType;
P1 : McPointType;
P0 : McPointType;
HOME : McPointType;
PZ : McPointType;
A : McAxisTargetType;

END_VAR

	PROGRAM _MAIN

	Feedrate(5000);    //move with reduced speed

	MoveA(A); //move HOME

//	MoveJ(P0);   //move to lower HOME pose

	MoveL(P1up); //move over the aim 1 pose
	Feedrate(2000);

	MoveL(P1);  //move to aim 1
	WaitTime(1);
	MoveL(P1up); //move over the aim 1 pose
	Feedrate(5000);
	MoveL(P2up); //move over the aim 2 pose
	Feedrate(2000);

	MoveL(P2);    //move to aim 2
	WaitTime(1);
	MoveL(P2up); //move over the aim 2 pose
	Feedrate(2000);

//	MoveL(P0);   //move to lower HOME pose
	MoveJ(HOME); //move to  HOME

END_PROGRAM
```

### Program Logical/File_explorer (IEC)

#### Types.typ
```iecst
TYPE
	TabInfo : 	STRUCT
		LastModified : ARRAY[0..49]OF DATE_AND_TIME;
		Type : ARRAY[0..49]OF MpFileManagerUIItemTypeEnum;
		Size : ARRAY[0..49]OF UDINT;
		Name : ARRAY[0..49]OF STRING[80];
		SelectedRow : USINT;
		NumberOfElements : USINT;
	END_STRUCT;
END_TYPE
```

#### Variables.var
```iecst
VAR
	iFile : INT;
	MpFileManagerUI_0 : MpFileManagerUI;
	MpFileMngSetup : MpFileManagerUISetupType;
	MpFileMngConnect : MpFileManagerUIConnectType;
	tabInfo : TabInfo;
END_VAR
```

#### Main.st
```iecst
PROGRAM _INIT
	(* Insert code here *)
	MpFileManagerUI_0(MpLink := ADR(gFileManagerUI), Enable :=1 , ErrorReset :=0 , UISetup :=MpFileMngSetup , UIConnect :=ADR(MpFileMngConnect));
	MpFileMngConnect.DeviceList.DeviceNames[0] := 'F';
END_PROGRAM

PROGRAM _CYCLIC
	(* Insert code here *)
	MpFileManagerUI_0();

	FOR iFile := 0 TO 49 BY 1 DO
		(* create arrays with file properties *)
		brsmemcpy(ADR(tabInfo.Name[iFile]), ADR(MpFileMngConnect.File.List.Items[iFile].Name), SIZEOF(tabInfo.Name[iFile]));
		brsmemcpy(ADR(tabInfo.Size[iFile]), ADR(MpFileMngConnect.File.List.Items[iFile].Size), SIZEOF(tabInfo.Size[iFile]));
		brsmemcpy(ADR(tabInfo.Type[iFile]), ADR(MpFileMngConnect.File.List.Items[iFile].ItemType), SIZEOF(tabInfo.Type[iFile]));
		brsmemcpy(ADR(tabInfo.LastModified[iFile]), ADR(MpFileMngConnect.File.List.Items[iFile].LastModified), SIZEOF(tabInfo.LastModified[iFile]));
		IF tabInfo.SelectedRow = iFile THEN
			MpFileMngConnect.File.List.Items[iFile].IsSelected := TRUE;
		END_IF
		(* numbers of elements in the table *)
		IF tabInfo.Type[iFile] <> mpFILE_ITEM_TYPE_NONE THEN
			tabInfo.NumberOfElements := tabInfo.NumberOfElements + 1;
		END_IF
	END_FOR

END_PROGRAM

PROGRAM _EXIT
	(* Insert code here *)
	 MpFileManagerUI_0.Enable := FALSE;
END_PROGRAM
```

### manulaTCP.st - not listed in the package file held
```iecst
#include 'Global.var'
VAR {AT 'Comau'}
X1 : LREAL;
Y1 : LREAL;
Z1 : LREAL;
A1 : LREAL;
B1 : LREAL;
C1 : LREAL;
END_VAR

	PROGRAM _MAIN
	Feedrate(3500);    //move with reduced speed
	PZ.Orient.Angle1 := A1;
	PZ.Orient.Angle3 := C1;
	PZ.Orient.Angle2 := B1;
	PZ.Pos.X := X1;
	PZ.Pos.Y := Y1;
	PZ.Pos.Z := Z1;
	MoveJ(PZ);

	END_PROGRAM
```

### Program Logical/Clock

#### Variables.var
```iecst
VAR
	TON_0 : TON;
	STEP : USINT := 0;
END_VAR
```

#### Main.st
```iecst
PROGRAM _INIT
	(* Insert code here *)

END_PROGRAM

PROGRAM _CYCLIC
	 CASE STEP OF
	0:
			TON_0( IN:=TRUE, PT:=T#1s200ms );
			IF TON_0.Q THEN
				STEP := 1;
			END_IF
	1:
			TON_0( IN:=FALSE, PT:=T#1s200ms );
			IF NOT TON_0.Q THEN
				STEP := 0;
			END_IF
	END_CASE
END_PROGRAM

PROGRAM _EXIT
	(* Insert code here *)

END_PROGRAM
```

### Program Logical/ComauAuto

#### Types.typ
```iecst
TYPE
	Step_typ :
		(
		ROBOTCTRL_DISABLED,
		ROBOTCTRL_POWER,
		ROBOTCTRL_WAIT_POWER,
		ROBOTCTRL_HOME,
		ROBOTCTRL_WAIT_HOME,
		ROBOTCTRL_READY,
		ROBOTCTRL_CALCULATE,
		ROBOTCTRL_CHECK,
		ROBOTCTRL_CALCULATE_P1,
		ROBOTCTRL_CALCULATE_P2,
		ROBOTCTRL_IS_MOVE_NEEDED,
		ROBOTCTRL_MOVE,
		ROBOTCTRL_ERROR_WRONG_AIM,
		ROBOTCTRL_ERROR,
		ROBOTCTRL_STOP,
		ROBOTCTRL_CONTINUE
		);
END_TYPE
```

#### Variables.var
```iecst
VAR
	RoboParameters : MpRoboArm6AxisParType;
	MpRoboArm6Axis_0 : MpRoboArm6Axis;
END_VAR
VAR CONSTANT
	SizeOfArray : INT := 13;
	IndexSize : INT := 3;
	Index : ARRAY[0..2] OF INT := [1,2,3];
END_VAR
VAR
	x : INT := 0;
	AimIsGood : BOOL := FALSE;
	Step : {REDUND_UNREPLICABLE} Step_typ := (0);
	cmdTurnOn : BOOL := FALSE;
	cmdTurnOff : BOOL := FALSE;
	cmdExecute : BOOL := FALSE;
	P1P2_Ok : BOOL := FALSE;
	cmdAck : BOOL;
	cmdStop : BOOL;
	cmdStart : BOOL;
	cmdContinue : BOOL;
END_VAR
```

#### Main.st
```iecst
PROGRAM _INIT

	MpRoboArm6Axis_0.Override  := 100.0;
	RoboParameters.CoordSystem := 0;
	RoboParameters.Velocity := 100;
	RoboParameters.Acceleration := 1000;
	RoboParameters.Deceleration := 1000;
	RoboParameters.ProgramName := 'Robotic.st';
	x;

END_PROGRAM

PROGRAM _CYCLIC

	RoboParameters.Jog.Velocity[0] := VelocityQ1;
	RoboParameters.Jog.Velocity[1] := VelocityQ2;
	RoboParameters.Jog.Velocity[2] := VelocityQ3;
	RoboParameters.Jog.Velocity[3] := VelocityQ4;
	RoboParameters.Jog.Velocity[4] := VelocityQ5;
	RoboParameters.Jog.Velocity[5] := VelocityQ6;

	IF cartezianVSjog THEN
		RoboParameters.Jog.CoordSystem := 10;
	ELSE
		RoboParameters.Jog.CoordSystem := 0;
	END_IF

	IF MpRoboArm6Axis_0.Error THEN
		Step := ROBOTCTRL_ERROR;
	END_IF;

	CASE Step OF

		ROBOTCTRL_DISABLED:
			IF cmdTurnOn THEN
				cmdTurnOn := FALSE;
				Step := ROBOTCTRL_POWER;
			END_IF;

		ROBOTCTRL_POWER:
			IF MpRoboArm6Axis_0.Info.ReadyToPowerOn THEN
				MpRoboArm6Axis_0.Power := TRUE;
				Step := ROBOTCTRL_WAIT_POWER;
			END_IF;

		ROBOTCTRL_WAIT_POWER:
			IF MpRoboArm6Axis_0.PowerOn THEN
				Step := ROBOTCTRL_HOME;
			END_IF;

		ROBOTCTRL_HOME:
			MpRoboArm6Axis_0.Home := TRUE;
			Step := ROBOTCTRL_WAIT_HOME;

		ROBOTCTRL_WAIT_HOME:
			IF MpRoboArm6Axis_0.IsHomed THEN
				MpRoboArm6Axis_0.Home := FALSE;
				Step := ROBOTCTRL_READY;
			END_IF;

		ROBOTCTRL_READY:
			IF cmdTurnOff THEN
				cmdTurnOff := FALSE;
				MpRoboArm6Axis_0.Power := FALSE;
			END_IF;

			IF NOT(MpRoboArm6Axis_0.PowerOn) THEN
				Step := ROBOTCTRL_DISABLED;
			END_IF;

			IF cmdExecute THEN
				cmdExecute:=FALSE;
				Step := ROBOTCTRL_CHECK; // if cmdexecute is active robot starts procedure

			END_IF;

		ROBOTCTRL_ERROR:
			// Error handling
			IF NOT(MpRoboArm6Axis_0.Error) THEN
				IF MpRoboArm6Axis_0.PowerOn THEN
					Step := ROBOTCTRL_READY;
				ELSE
					Step := ROBOTCTRL_DISABLED;
				END_IF;
			END_IF;

		ROBOTCTRL_CHECK: 	//checking if aim targets are available
			AimIsGood:=TRUE;
			FOR x:=0  TO SizeOfArray DO
				pom[0]:=1;
				IF gAimPos[x]>0 THEN
					pom[1]:=1;
					IF (gIsPosGood[x]=FALSE) THEN
						pom[2]:=1;
						Step:=ROBOTCTRL_ERROR_WRONG_AIM;
						AimIsGood:=0;
					END_IF;
				END_IF;
			END_FOR;
			IF AimIsGood=TRUE THEN

				y:=0;
				Step:=ROBOTCTRL_CALCULATE;

			END_IF;

		ROBOTCTRL_CALCULATE:
			//checking if any move is needed and if all moves are done
			IF	P1P2_Ok THEN
				Step:=ROBOTCTRL_IS_MOVE_NEEDED;
			ELSIF y<IndexSize THEN
				Step:=ROBOTCTRL_CALCULATE_P1;
			ELSE
				cmdExecute:=FALSE;
				Step:=ROBOTCTRL_READY;
			END_IF;

		ROBOTCTRL_CALCULATE_P1:
			//assigning values to P1 and P1up
			FOR x:=0  TO SizeOfArray DO
				IF gActPos[x]=Index[y] THEN
					pom[3]:=1;
					P1.Orient.Angle1:=gRobPos[x].Orient.Angle1;
					P1.Orient.Angle2:=gRobPos[x].Orient.Angle2;
					P1.Orient.Angle3:=gRobPos[x].Orient.Angle3;
					P1.Pos.X:=gRobPos[x].Pos.X;
					P1.Pos.Y:=gRobPos[x].Pos.Y;
					P1.Pos.Z:=gRobPos[x].Pos.Z;
					P1up.Orient.Angle1:=gRobPos[x].Orient.Angle1;
					P1up.Orient.Angle2:=gRobPos[x].Orient.Angle2;
					P1up.Orient.Angle3:=gRobPos[x].Orient.Angle3;
					P1up.Pos.X:=gRobPos[x].Pos.X;
					P1up.Pos.Y:=gRobPos[x].Pos.Y;
					P1up.Pos.Z:=gRobPos[x].Pos.Z+100;

				END_IF;
			END_FOR;
			Step:=ROBOTCTRL_CALCULATE_P2;

		ROBOTCTRL_CALCULATE_P2:
				//assigning values to P2 and P2up
			FOR x:=0  TO SizeOfArray DO
				IF gAimPos[x]=Index[y] THEN
					pom[4]:=1;
					P2.Orient.Angle1:=gRobPos[x].Orient.Angle1;
					P2.Orient.Angle2:=gRobPos[x].Orient.Angle2;
					P2.Orient.Angle3:=gRobPos[x].Orient.Angle3;
					P2.Pos.X:=gRobPos[x].Pos.X;
					P2.Pos.Y:=gRobPos[x].Pos.Y;
					P2.Pos.Z:=gRobPos[x].Pos.Z;
					P2up.Orient.Angle1:=gRobPos[x].Orient.Angle1;
					P2up.Orient.Angle2:=gRobPos[x].Orient.Angle2;
					P2up.Orient.Angle3:=gRobPos[x].Orient.Angle3;
					P2up.Pos.X:=gRobPos[x].Pos.X;
					P2up.Pos.Y:=gRobPos[x].Pos.Y;
					P2up.Pos.Z:=gRobPos[x].Pos.Z+100;

				END_IF;
			END_FOR;
			P1P2_Ok:=1; // this flag means that new P1 and new P2 have been assigned
			Step:=ROBOTCTRL_CALCULATE;

		ROBOTCTRL_IS_MOVE_NEEDED:
			//checking if actual and aim positions are not the same
			IF P1.Orient.Angle1=P2.Orient.Angle1 AND P1.Pos.X=P2.Pos.X AND P1.Orient.Angle2=P2.Orient.Angle2 AND P1.Pos.Y=P2.Pos.Y AND P1.Orient.Angle3=P2.Orient.Angle3 AND P1.Pos.Z=P2.Pos.Z THEN
				y:=y+1;
				P1P2_Ok:=0;
				Step:=ROBOTCTRL_CALCULATE;
			ELSE
				Step:=ROBOTCTRL_MOVE;
			END_IF;

		ROBOTCTRL_MOVE:
			IF cmdTurnOff THEN
				cmdTurnOff := FALSE;
				MpRoboArm6Axis_0.Power := FALSE;
				Step:=ROBOTCTRL_DISABLED;
			END_IF;

			IF cmdStop OR MpRoboArm6Axis_0.MoveInterrupted THEN
				cmdStop := FALSE;
				Step:=ROBOTCTRL_STOP;
			END_IF;

			//executing move procedure
			MpRoboArm6Axis_0.MoveProgram:=1;
			IF MpRoboArm6Axis_0.MoveDone THEN
				MpRoboArm6Axis_0.MoveProgram:=0;
				y:=y+1;
				P1P2_Ok:=0;
				Step:=ROBOTCTRL_CALCULATE;
			END_IF

		ROBOTCTRL_STOP:
			MpRoboArm6Axis_0.Interrupt:=TRUE;
			IF cmdContinue THEN
				cmdContinue:=FALSE;
				MpRoboArm6Axis_0.Interrupt:=FALSE;
				Step:=ROBOTCTRL_CONTINUE;
			END_IF

		ROBOTCTRL_CONTINUE:
			MpRoboArm6Axis_0.Continue:=1;
			IF  MpRoboArm6Axis_0.InMotion THEN
				MpRoboArm6Axis_0.Continue:=0;
				Step:=ROBOTCTRL_MOVE;
			END_IF

		ROBOTCTRL_ERROR_WRONG_AIM:
			//handling wrong target error
			IF cmdAck THEN
				cmdAck:=FALSE;
				Step:=ROBOTCTRL_READY;
			END_IF;

	END_CASE;

	MpRoboArm6Axis_0.MpLink     := ADR(gAxesGroup_Racer3_1);
	MpRoboArm6Axis_0.Parameters := ADR(RoboParameters);
	MpRoboArm6Axis_0.Override := 100.0;
	MpRoboArm6Axis_0.Enable := TRUE;
	MpRoboArm6Axis_0();

END_PROGRAM

PROGRAM _EXIT
				(* Insert code here *)

				END_PROGRAM
```

### Program Logical/ElementsDetection

#### Types.typ
```iecst
TYPE
	PixelCounterLimits : 	STRUCT
		WrenchLimit : UDINT;
		WasherBoltLimit : UDINT;
		ScrewLimit : UDINT;
		HolderLimit : UDINT;
	END_STRUCT;
	CameraStruct : 	STRUCT
		ExposureTime : UDINT := 30000;
		Focus : UINT := 30000;
		NumSearch : USINT;
		Enable : BOOL;
		diTrigger : BOOL;
		ImageAcq : BOOL;
		PixelCntSquareArray : ARRAY[0..13]OF UDINT;
		Ready : BOOL;
		FlashColor : USINT;
		ModelNumArray : ARRAY[0..13]OF USINT;
		FlashSegment : USINT;
	END_STRUCT;
END_TYPE
```

#### Variables.var
```iecst
VAR
	i : USINT;
	PixelRange_0 : PixelCounterLimits;
	DetectedSquares : USINT;
	Camera_0 : CameraStruct;
END_VAR
```

#### Main.st
```iecst
PROGRAM _INIT
	//CAMERA INITIAL VALUES
	Camera_0.Focus := 30000;
	Camera_0.ExposureTime := 40000;
	Camera_0.NumSearch := 14;
	Camera_0.Enable := 1;

	PixelRange_0.ScrewLimit := 200;
	PixelRange_0.WasherBoltLimit := 500;
	PixelRange_0.WrenchLimit := 2000;
	PixelRange_0.HolderLimit := 10000;

	///////////////////////////////
	DetectedSquares := 7;
	//////////////////////////////

END_PROGRAM

PROGRAM _CYCLIC
	//IMAGE ACQUISITION
	Camera_0.ImageAcq := Camera_0.diTrigger AND Camera_0.Ready;

	DetectedSquares := 0;

	FOR i := 0 TO 13 DO
		//SQUARES DETECTION
		SquareArray[Camera_0.ModelNumArray[i]-1] := Camera_0.PixelCntSquareArray[i] < PixelRange_0.HolderLimit;
		IF Camera_0.PixelCntSquareArray[i] < PixelRange_0.HolderLimit THEN
			DetectedSquares := DetectedSquares + 1;
		END_IF

		IF Camera_0.PixelCntSquareArray[i] < 50 THEN
			//NOTHING
			ElementsArray[Camera_0.ModelNumArray[i]-1] := 0;
		ELSIF Camera_0.PixelCntSquareArray[i] < PixelRange_0.ScrewLimit THEN
			//SCREW
			//index nietestowy := 1
			ElementsArray[Camera_0.ModelNumArray[i]-1] := 1;
		ELSIF Camera_0.PixelCntSquareArray[i] < PixelRange_0.WasherBoltLimit THEN
			//WASHER BOLT
			//index nietestowy := 2
			ElementsArray[Camera_0.ModelNumArray[i]-1] := 2;
		ELSIF Camera_0.PixelCntSquareArray[i] < PixelRange_0.WrenchLimit THEN
			//WRENCH
			//index nietestowy := 4
			ElementsArray[Camera_0.ModelNumArray[i]-1] := 4;
		ELSE
			ElementsArray[Camera_0.ModelNumArray[i]-1] := 0;
		END_IF;

	END_FOR;

END_PROGRAM

PROGRAM _EXIT

END_PROGRAM
```

### Program Logical/PackML_Auto

#### Main.st
```iecst
PROGRAM _INIT
	(* Insert code here *)

END_PROGRAM

PROGRAM _CYCLIC
	Starting;
	Idle;
	Stopping;
	Resetting;
	Execute;
	Completing;
	Complete;
	Stopped;
END_PROGRAM

PROGRAM _EXIT
	(* Insert code here *)

END_PROGRAM
```

#### Stopped.st
```iecst
ACTION Stopped:
	IF MpPackMLStateIsActive(gPackMLCore,
		mpPACKML_STATE_STOPPED,
		1) THEN

		//MpPackMLMode_Auto.Reset := 0;

		IF diReset THEN
			MpPackMLStateComplete(gPackMLCore, 1);
		ELSIF toAbort THEN
			MpPackMLAbort(gPackMLCore, 1);
		END_IF

	END_IF

END_ACTION
```

#### Stopping.st
```iecst
ACTION Stopping:
	IF MpPackMLStateIsActive(gPackMLCore,
		mpPACKML_STATE_STOPPING,
		1) THEN

		test := 100;
		//STOP EVERYTHING

		IF toStopped THEN
		//	MpPackMLStateComplete(gPackMLCore, 1);
			MpPackMLMode_Auto.StateComplete := 1;
		ELSIF toAbort THEN
			MpPackMLAbort(gPackMLCore, 1);
		END_IF

		END_IF

END_ACTION
```

### Program Logical/PackML_Logic

#### Main.st
```iecst
PROGRAM _INIT
	MpPackMLCore_0.MpLink := ADR(gPackMLCore);
	MpPackMLCore_0.Enable := TRUE;

	MpPackMLMode_Auto.MpLink := ADR(gPackMLCore);
	MpPackMLMode_Auto.Enable := TRUE;
	MpPackMLMode_Auto.ModeID := 1;

	MpPackMLMode_SemiAuto.MpLink := ADR(gPackMLCore);
	MpPackMLMode_SemiAuto.Enable := TRUE;
	MpPackMLMode_SemiAuto.ModeID := 2;

	MpPackMLMode_Manual.MpLink := ADR(gPackMLCore);
	MpPackMLMode_Manual.Enable := TRUE;
	MpPackMLMode_Manual.ModeID := 3;

	//ACTIVATE := 1 ?????

END_PROGRAM

PROGRAM _CYCLIC
	MpPackMLCore_0();
	MpPackMLMode_Auto();
	MpPackMLMode_SemiAuto();
	MpPackMLMode_Manual();

END_PROGRAM

PROGRAM _EXIT
	MpPackMLCore_0.Enable := 0;
	MpPackMLMode_Auto.Enable := 0;
	MpPackMLMode_SemiAuto.Enable := 0;
	MpPackMLMode_Manual.Enable := 0;

	MpPackMLCore_0();
	MpPackMLMode_Auto();
	MpPackMLMode_SemiAuto();
	MpPackMLMode_Manual();

	diReset;
	diStop;
	toStopped;
	test;

END_PROGRAM
```

### Program Logical/Podstawki

#### Variables.var
```iecst
VAR
	ExposureTime : UDINT := 30000;
	Focus : UINT := 30000;
	NumSearch : USINT;
	Enable : BOOL;
	diTrigger : BOOL;
	ImageAcq : BOOL;
	i : USINT;
END_VAR
```

#### Main.st
```iecst
PROGRAM _INIT
	(* Insert code here *)
	Focus := 30000;
	ExposureTime := 30000;
	NumSearch := 14;
	Enable := 1;

END_PROGRAM

PROGRAM _CYCLIC
	(* Insert code here *)

	ImageAcq := diTrigger AND CameraReady;

	FOR i := 0 TO 13 DO
		IF PixelCntArray[i] < 10000 THEN
			SquareArray[i] := 0;
		ELSE
			SquareArray[i] := 1;
		END_IF;

	END_FOR;

	PixelCntArray;
	ResetAcq;
	FlashColor;
	FlashSegment;

END_PROGRAM

PROGRAM _EXIT
	(* Insert code here *)

END_PROGRAM
```

### Program Logical/Program

#### Main.st
```iecst
PROGRAM _INIT
	(* Insert code here *)

END_PROGRAM

PROGRAM _CYCLIC
	(* Insert code here *)
	gCamera;

END_PROGRAM

PROGRAM _EXIT
	(* Insert code here *)

END_PROGRAM
```

### Program Logical/Recipe

#### Variables.var
```iecst
VAR
	clear : BOOL;
	MpRecipeXml_0 : MpRecipeXml;
	name : STRING[80];
	ScrewWasher : BOOL;
	Wrench : BOOL;
	Screw : BOOL;
	MpRecipeRegPar_0 : MpRecipeRegPar;
	ScrewPosible : BOOL;
	WrenchPosible : BOOL;
	ScrewWasherPosible : BOOL;
	i : INT;
END_VAR
```

#### Main.st
```iecst
PROGRAM _INIT
	(* Insert code here *)
	MpRecipeXml_0.MpLink := ADR(gRecipeXml);
	MpRecipeXml_0.Enable := TRUE;

	MpRecipeRegPar_0.MpLink := ADR(gRecipeXml);
	MpRecipeRegPar_0.Enable := TRUE;
	gAimPos;
	ScrewPosible := TRUE;
	ScrewWasherPosible := TRUE;
	WrenchPosible := TRUE;
	name;
END_PROGRAM

PROGRAM _CYCLIC
	(* Insert code here *)

	IF clear THEN

		FOR i := 0 TO 13 BY 1 DO
		gAimPos[i] :=0 ;
		END_FOR;

		ScrewPosible := TRUE;
		ScrewWasherPosible := TRUE;
		WrenchPosible := TRUE;
	END_IF

	FOR i := 0 TO 13 BY 1 DO

		IF gAimPos[i]  = 1 THEN
			ScrewPosible := FALSE;
		END_IF
		IF gAimPos[i]  = 2 THEN
			ScrewWasherPosible := FALSE;
		END_IF
		IF gAimPos[i]  = 4 THEN
			WrenchPosible := FALSE;
		END_IF

	END_FOR;

	MpRecipeXml_0();
	MpRecipeXml_0.DeviceName := ADR('RecipeDir');

	MpRecipeRegPar_0();
	MpRecipeRegPar_0.PVName := ADR('gAimPos');

	MpRecipeXml_0.FileName := ADR(name);

END_PROGRAM

PROGRAM _EXIT
	(* Insert code here *)

END_PROGRAM
```

Listed in the project but not available here: Logical/PackML/PackML_Logic, Logical/PackML/PackML_Auto/Types.typ, Logical/Sources/OpcCtrl
